LIN {X 0,Y 208.668,Z 381.617,A -85,B 0,C 180,E1 -22016.518,E2 -22016.518} C_VEL
LIN {X 0,Y 207.654,Z 387.475,A -85,B 0,C 180,E1 -22016.591,E2 -22016.591} C_VEL
LIN {X 0,Y 204.493,Z 399.145,A -85,B 0,C 180,E1 -22016.563,E2 -22016.563} C_VEL
LIN {X 0,Y 203.408,Z 405.081,A -85,B 0,C 180,E1 -22016.629,E2 -22016.629} C_VEL
LIN {X 0,Y 203.257,Z 407.077,A -85,B 0,C 180,E1 -22016.685,E2 -22016.685} C_VEL
LIN {X 0,Y 201.605,Z 442.654,A -85,B 0,C 180,E1 -22017.92,E2 -22017.92} C_VEL
LIN {X 0,Y 200.293,Z 456.074,A -85,B 0,C 180,E1 -22018.76,E2 -22018.76} C_VEL
LIN {X 0,Y 198.653,Z 468.006,A -85,B 0,C 180,E1 -22019.874,E2 -22019.874} C_VEL
LIN {X 0,Y 196.505,Z 480.066,A -85,B 0,C 180,E1 -22021.424,E2 -22021.424} C_VEL
LIN {X 0,Y 193.917,Z 491.578,A -85,B 0,C 180,E1 -22023.354,E2 -22023.354} C_VEL
LIN {X 0,Y 191.601,Z 501.991,A -85,B 0,C 180,E1 -22025.63,E2 -22025.63} C_VEL
LIN {X 0,Y 189.316,Z 511.311,A -85,B 0,C 180,E1 -22028.21,E2 -22028.21} C_VEL
LIN {X 0,Y 187.461,Z 518.995,A -85,B 0,C 180,E1 -22030.852,E2 -22030.852} C_VEL
LIN {X 0,Y 185.631,Z 526.51,A -85,B 0,C 180,E1 -22034.07,E2 -22034.07} C_VEL
LIN {X 0,Y 184.166,Z 533.424,A -85,B 0,C 180,E1 -22037.886,E2 -22037.886} C_VEL
LIN {X 0,Y 183.486,Z 537.971,A -85,B 0,C 180,E1 -22041.188,E2 -22041.188} C_VEL
LIN {X 0,Y 183.285,Z 540.362,A -85,B 0,C 180,E1 -22043.396,E2 -22043.396} C_VEL
LIN {X 0,Y 183.153,Z 542.708,A -85,B 0,C 180,E1 -22046.1,E2 -22046.1} C_VEL
LIN {X 0,Y 183.324,Z 544.894,A -85,B 0,C 180,E1 -22050.001,E2 -22050.001} C_VEL
LIN {X 0,Y 183.072,Z 545.742,A -85,B 0,C 180,E1 -22053.507,E2 -22053.507} C_VEL
LIN {X 0,Y 183.214,Z 545.668,A -85,B 0,C 180,E1 -22056.609,E2 -22056.609} C_VEL
LIN {X 0,Y 184.032,Z 544.175,A -85,B 0,C 180,E1 -22061.009,E2 -22061.009} C_VEL
LIN {X 0,Y 185.663,Z 541.115,A -85,B 0,C 180,E1 -22065.366,E2 -22065.366} C_VEL
LIN {X 0,Y 187.738,Z 537.669,A -85,B 0,C 180,E1 -22068.555,E2 -22068.555} C_VEL
LIN {X 0,Y 190.309,Z 533.167,A -85,B 0,C 180,E1 -22071.673,E2 -22071.673} C_VEL
LIN {X 0,Y 193.539,Z 527.136,A -85,B 0,C 180,E1 -22074.873,E2 -22074.873} C_VEL
LIN {X 0,Y 196.958,Z 520.396,A -85,B 0,C 180,E1 -22077.638,E2 -22077.638} C_VEL
LIN {X 0,Y 201.249,Z 511.587,A -85,B 0,C 180,E1 -22080.423,E2 -22080.423} C_VEL
LIN {X 0,Y 205.142,Z 502.581,A -85,B 0,C 180,E1 -22082.656,E2 -22082.656} C_VEL
LIN {X 0,Y 208.987,Z 492.681,A -85,B 0,C 180,E1 -22084.576,E2 -22084.576} C_VEL
LIN {X 0,Y 212.638,Z 481.706,A -85,B 0,C 180,E1 -22086.214,E2 -22086.214} C_VEL
LIN {X 0,Y 215.466,Z 471.415,A -85,B 0,C 180,E1 -22087.41,E2 -22087.41} C_VEL
LIN {X 0,Y 218.344,Z 458.36,A -85,B 0,C 180,E1 -22088.522,E2 -22088.522} C_VEL
LIN {X 0,Y 220.277,Z 445.531,A -85,B 0,C 180,E1 -22089.282,E2 -22089.282} C_VEL
LIN {X 0,Y 221.553,Z 429.787,A -85,B 0,C 180,E1 -22089.834,E2 -22089.834} C_VEL
LIN {X 0,Y 223.363,Z 398.956,A -85,B 0,C 180,E1 -22090.749,E2 -22090.749} C_VEL
LIN {X 0,Y 222.537,Z 393.348,A -85,B 0,C 180,E1 -22091.214,E2 -22091.214} C_VEL
LIN {X 0,Y 216.187,Z 378.63,A -85,B 0,C 180,E1 -22093.651,E2 -22093.651} C_VEL
LIN {X 0,Y 210.751,Z 367.719,A -85,B 0,C 180,E1 -22095.876,E2 -22095.876} C_VEL
LIN {X 0,Y 204.884,Z 357.45,A -85,B 0,C 180,E1 -22098.458,E2 -22098.458} C_VEL
LIN {X 0,Y 201.95,Z 352.743,A -85,B 0,C 180,E1 -22099.843,E2 -22099.843} C_VEL
LIN {X 0,Y 198.712,Z 347.595,A -85,B 0,C 180,E1 -22101.478,E2 -22101.478} C_VEL
LIN {X 0,Y 195.305,Z 342.411,A -85,B 0,C 180,E1 -22103.324,E2 -22103.324} C_VEL
LIN {X 0,Y 191.41,Z 336.757,A -85,B 0,C 180,E1 -22105.63,E2 -22105.63} C_VEL
LIN {X 0,Y 187.73,Z 332.249,A -85,B 0,C 180,E1 -22108,E2 -22108} C_VEL
LIN {X 0,Y 186.391,Z 329.867,A -85,B 0,C 180,E1 -22109.087,E2 -22109.087} C_VEL
LIN {X 0,Y 185.613,Z 327.361,A -85,B 0,C 180,E1 -22111.905,E2 -22111.905} C_VEL
LIN {X 0,Y 185.59,Z 327.368,A -85,B 0,C 180,E1 -22115.383,E2 -22115.383} C_VEL
LIN {X 0,Y 185.677,Z 327.344,A -85,B 0,C 180,E1 -22121.133,E2 -22121.133} C_VEL
LIN {X 0,Y 185.697,Z 327.342,A -85,B 0,C 180,E1 -22124.637,E2 -22124.637} C_VEL
LIN {X 0,Y 185.891,Z 327.313,A -85,B 0,C 180,E1 -22129.417,E2 -22129.417} C_VEL
LIN {X 0,Y 185.953,Z 327.306,A -85,B 0,C 180,E1 -22133.489,E2 -22133.489} C_VEL
LIN {X 0,Y 186.208,Z 327.274,A -85,B 0,C 180,E1 -22137.837,E2 -22137.837} C_VEL
LIN {X 0,Y 186.406,Z 327.249,A -85,B 0,C 180,E1 -22140,E2 -22140} C_VEL
LIN {X 0,Y 185.924,Z 327.309,A -85,B 0,C 180,E1 -22144.335,E2 -22144.335} C_VEL
LIN {X 0,Y 186.011,Z 327.3,A -85,B 0,C 180,E1 -22148.692,E2 -22148.692} C_VEL
LIN {X 0,Y 185.736,Z 327.337,A -85,B 0,C 180,E1 -22153.122,E2 -22153.122} C_VEL
LIN {X 0,Y 185.691,Z 327.346,A -85,B 0,C 180,E1 -22157.625,E2 -22157.625} C_VEL
LIN {X 0,Y 185.604,Z 327.548,A -85,B 0,C 180,E1 -22160.865,E2 -22160.865} C_VEL
LIN {X 0,Y 186.322,Z 329.769,A -85,B 0,C 180,E1 -22161.505,E2 -22161.505} C_VEL
LIN {X 0,Y 188.182,Z 332.015,A -85,B 0,C 180,E1 -22162.797,E2 -22162.797} C_VEL
LIN {X 0,Y 190.075,Z 333.259,A -85,B 0,C 180,E1 -22163.952,E2 -22163.952} C_VEL
LIN {X 0,Y 191.863,Z 336.387,A -85,B 0,C 180,E1 -22165.13,E2 -22165.13} C_VEL
LIN {X 0,Y 194.423,Z 338.858,A -85,B 0,C 180,E1 -22166.572,E2 -22166.572} C_VEL
LIN {X 0,Y 196.875,Z 342.368,A -85,B 0,C 180,E1 -22167.939,E2 -22167.939} C_VEL
LIN {X 0,Y 198.391,Z 344.088,A -85,B 0,C 180,E1 -22168.715,E2 -22168.715} C_VEL
LIN {X 0,Y 202.124,Z 349.183,A -85,B 0,C 180,E1 -22170.565,E2 -22170.565} C_VEL
LIN {X 0,Y 207.219,Z 356.189,A -85,B 0,C 180,E1 -22172.864,E2 -22172.864} C_VEL
LIN {X 0,Y 214.375,Z 367.343,A -85,B 0,C 180,E1 -22175.802,E2 -22175.802} C_VEL
LIN {X 0,Y 218.893,Z 375.323,A -85,B 0,C 180,E1 -22177.519,E2 -22177.519} C_VEL
LIN {X 0,Y 223.957,Z 386.107,A -85,B 0,C 180,E1 -22179.382,E2 -22179.382} C_VEL
LIN {X 0,Y 221.263,Z 429.958,A -85,B 0,C 180,E1 -22180.737,E2 -22180.737} C_VEL
LIN {X 0,Y 219.571,Z 443.344,A -85,B 0,C 180,E1 -22181.471,E2 -22181.471} C_VEL
LIN {X 0,Y 217.663,Z 453.695,A -85,B 0,C 180,E1 -22182.29,E2 -22182.29} C_VEL
LIN {X 0,Y 215.148,Z 465.009,A -85,B 0,C 180,E1 -22183.519,E2 -22183.519} C_VEL
LIN {X 0,Y 212.177,Z 475.253,A -85,B 0,C 180,E1 -22184.926,E2 -22184.926} C_VEL
LIN {X 0,Y 208.834,Z 485.292,A -85,B 0,C 180,E1 -22186.709,E2 -22186.709} C_VEL
LIN {X 0,Y 205.109,Z 494.662,A -85,B 0,C 180,E1 -22188.796,E2 -22188.796} C_VEL
LIN {X 0,Y 200.69,Z 504.369,A -85,B 0,C 180,E1 -22191.567,E2 -22191.567} C_VEL
LIN {X 0,Y 196.696,Z 512.209,A -85,B 0,C 180,E1 -22194.505,E2 -22194.505} C_VEL
LIN {X 0,Y 193.786,Z 517.529,A -85,B 0,C 180,E1 -22197.043,E2 -22197.043} C_VEL
LIN {X 0,Y 190.747,Z 522.64,A -85,B 0,C 180,E1 -22200.171,E2 -22200.171} C_VEL
LIN {X 0,Y 187.947,Z 527.003,A -85,B 0,C 180,E1 -22203.824,E2 -22203.824} C_VEL
LIN {X 0,Y 185.701,Z 530.147,A -85,B 0,C 180,E1 -22207.761,E2 -22207.761} C_VEL
LIN {X 0,Y 184.78,Z 531.287,A -85,B 0,C 180,E1 -22209.981,E2 -22209.981} C_VEL
LIN {X 0,Y 183.972,Z 532.088,A -85,B 0,C 180,E1 -22212.752,E2 -22212.752} C_VEL
LIN {X 0,Y 183.211,Z 532.19,A -85,B 0,C 180,E1 -22216.692,E2 -22216.692} C_VEL
LIN {X 0,Y 183.023,Z 531.678,A -85,B 0,C 180,E1 -22218.93,E2 -22218.93} C_VEL
LIN {X 0,Y 183,Z 530.746,A -85,B 0,C 180,E1 -22221.162,E2 -22221.162} C_VEL
LIN {X 0,Y 183.409,Z 528.14,A -85,B 0,C 180,E1 -22225.057,E2 -22225.057} C_VEL
LIN {X 0,Y 183.952,Z 524.248,A -85,B 0,C 180,E1 -22228.904,E2 -22228.904} C_VEL
LIN {X 0,Y 184.943,Z 519.717,A -85,B 0,C 180,E1 -22232.177,E2 -22232.177} C_VEL
LIN {X 0,Y 186.489,Z 512.867,A -85,B 0,C 180,E1 -22235.947,E2 -22235.947} C_VEL
LIN {X 0,Y 188.412,Z 505.439,A -85,B 0,C 180,E1 -22239.12,E2 -22239.12} C_VEL
LIN {X 0,Y 190.372,Z 497.865,A -85,B 0,C 180,E1 -22241.714,E2 -22241.714} C_VEL
LIN {X 0,Y 192.63,Z 488.695,A -85,B 0,C 180,E1 -22244.256,E2 -22244.256} C_VEL
LIN {X 0,Y 194.994,Z 478.471,A -85,B 0,C 180,E1 -22246.488,E2 -22246.488} C_VEL
LIN {X 0,Y 197.452,Z 467.103,A -85,B 0,C 180,E1 -22248.413,E2 -22248.413} C_VEL
LIN {X 0,Y 199.305,Z 455.369,A -85,B 0,C 180,E1 -22249.973,E2 -22249.973} C_VEL
LIN {X 0,Y 200.678,Z 442.511,A -85,B 0,C 180,E1 -22251.237,E2 -22251.237} C_VEL
LIN {X 0,Y 201.914,Z 429.718,A -85,B 0,C 180,E1 -22252.039,E2 -22252.039} C_VEL
LIN {X 0,Y 203.605,Z 395.641,A -85,B 0,C 180,E1 -22253.214,E2 -22253.214} C_VEL
LIN {X 0,Y 204.769,Z 366.988,A -85,B 0,C 180,E1 -22254.17,E2 -22254.17} C_VEL
LIN {X 0,Y 200.862,Z 356.621,A -85,B 0,C 180,E1 -22255.245,E2 -22255.245} C_VEL
LIN {X 0,Y 193.205,Z 341.376,A -85,B 0,C 180,E1 -22257.295,E2 -22257.295} C_VEL
LIN {X 0,Y 187.089,Z 330.978,A -85,B 0,C 180,E1 -22259.007,E2 -22259.007} C_VEL
LIN {X 0,Y 185.79,Z 328.546,A -85,B 0,C 180,E1 -22259.4,E2 -22259.4} C_VEL
LIN {X 0,Y 185.544,Z 327.369,A -85,B 0,C 180,E1 -22259.575,E2 -22259.575} C_VEL
LIN {X 0,Y 185.494,Z 327.378,A -85,B 0,C 180,E1 -22264.631,E2 -22264.631} C_VEL
LIN {X 0,Y 185.497,Z 327.373,A -85,B 0,C 180,E1 -22267.313,E2 -22267.313} C_VEL
LIN {X 0,Y 185.458,Z 327.383,A -85,B 0,C 180,E1 -22270.72,E2 -22270.72} C_VEL
LIN {X 0,Y 185.454,Z 327.379,A -85,B 0,C 180,E1 -22276.054,E2 -22276.054} C_VEL
LIN {X 0,Y 185.462,Z 327.371,A -85,B 0,C 180,E1 -22279.894,E2 -22279.894} C_VEL
LIN {X 0,Y 185.501,Z 327.364,A -85,B 0,C 180,E1 -22282.711,E2 -22282.711} C_VEL
LIN {X 0,Y 185.537,Z 327.362,A -85,B 0,C 180,E1 -22287.974,E2 -22287.974} C_VEL
LIN {X 0,Y 185.575,Z 327.347,A -85,B 0,C 180,E1 -22290.576,E2 -22290.576} C_VEL
LIN {X 0,Y 185.575,Z 327.37,A -85,B 0,C 180,E1 -22295.381,E2 -22295.381} C_VEL
LIN {X 0,Y 185.668,Z 327.34,A -85,B 0,C 180,E1 -22301.134,E2 -22301.134} C_VEL
LIN {X 0,Y 185.689,Z 327.354,A -85,B 0,C 180,E1 -22304.637,E2 -22304.637} C_VEL
LIN {X 0,Y 185.883,Z 327.307,A -85,B 0,C 180,E1 -22309.419,E2 -22309.419} C_VEL
LIN {X 0,Y 185.934,Z 327.319,A -85,B 0,C 180,E1 -22313.489,E2 -22313.489} C_VEL
LIN {X 0,Y 186.198,Z 327.283,A -85,B 0,C 180,E1 -22317.837,E2 -22317.837} C_VEL
LIN {X 0,Y 186.398,Z 327.242,A -85,B 0,C 180,E1 -22320,E2 -22320} C_VEL
LIN {X 0,Y 185.917,Z 327.323,A -85,B 0,C 180,E1 -22324.336,E2 -22324.336} C_VEL
LIN {X 0,Y 186.003,Z 327.303,A -85,B 0,C 180,E1 -22328.693,E2 -22328.693} C_VEL
LIN {X 0,Y 185.729,Z 327.338,A -85,B 0,C 180,E1 -22333.123,E2 -22333.123} C_VEL
LIN {X 0,Y 185.685,Z 327.35,A -85,B 0,C 180,E1 -22337.626,E2 -22337.626} C_VEL
LIN {X 0,Y 185.592,Z 327.363,A -85,B 0,C 180,E1 -22342.252,E2 -22342.252} C_VEL
LIN {X 0,Y 185.558,Z 327.37,A -85,B 0,C 180,E1 -22347.033,E2 -22347.033} C_VEL
LIN {X 0,Y 185.575,Z 327.368,A -85,B 0,C 180,E1 -22349.494,E2 -22349.494} C_VEL
LIN {X 0,Y 185.507,Z 327.38,A -85,B 0,C 180,E1 -22354.631,E2 -22354.631} C_VEL
LIN {X 0,Y 185.541,Z 327.375,A -85,B 0,C 180,E1 -22357.305,E2 -22357.305} C_VEL
LIN {X 0,Y 185.481,Z 327.384,A -85,B 0,C 180,E1 -22360.731,E2 -22360.731} C_VEL
LIN {X 0,Y 185.456,Z 327.387,A -85,B 0,C 180,E1 -22366.057,E2 -22366.057} C_VEL
LIN {X 0,Y 185.503,Z 327.579,A -85,B 0,C 180,E1 -22367.706,E2 -22367.706} C_VEL
LIN {X 0,Y 186.847,Z 332.585,A -85,B 0,C 180,E1 -22370.517,E2 -22370.517} C_VEL
LIN {X 0,Y 193.158,Z 346.017,A -85,B 0,C 180,E1 -22372.399,E2 -22372.399} C_VEL
LIN {X 0,Y 200.302,Z 363.714,A -85,B 0,C 180,E1 -22374.448,E2 -22374.448} C_VEL
LIN {X 0,Y 201.381,Z 367.117,A -85,B 0,C 180,E1 -22374.772,E2 -22374.772} C_VEL
LIN {X 0,Y 203.856,Z 392.612,A -85,B 0,C 180,E1 -22376.204,E2 -22376.204} C_VEL
LIN {X 0,Y 203.257,Z 407.077,A -85,B 0,C 180,E1 -22376.685,E2 -22376.685} C_VEL
LIN {X 0,Y 202.421,Z 412.922,A -85,B 0,C 180,E1 -22376.783,E2 -22376.783} C_VEL
LIN {X 0,Y 196.521,Z 431.869,A -85,B 0,C 180,E1 -22376.609,E2 -22376.609} C_VEL
LIN {X 0,Y 195.694,Z 437.696,A -85,B 0,C 180,E1 -22376.747,E2 -22376.747} C_VEL
LIN {X 0,Y 194.622,Z 450.72,A -85,B 0,C 180,E1 -22377.435,E2 -22377.435} C_VEL
LIN {X 0,Y 192.985,Z 462.95,A -85,B 0,C 180,E1 -22378.435,E2 -22378.435} C_VEL
LIN {X 0,Y 191.223,Z 473.552,A -85,B 0,C 180,E1 -22379.647,E2 -22379.647} C_VEL
LIN {X 0,Y 188.881,Z 485.038,A -85,B 0,C 180,E1 -22381.378,E2 -22381.378} C_VEL
LIN {X 0,Y 186.426,Z 495.503,A -85,B 0,C 180,E1 -22383.407,E2 -22383.407} C_VEL
LIN {X 0,Y 184.119,Z 505.106,A -85,B 0,C 180,E1 -22385.776,E2 -22385.776} C_VEL
LIN {X 0,Y 181.706,Z 514.437,A -85,B 0,C 180,E1 -22388.669,E2 -22388.669} C_VEL
LIN {X 0,Y 179.712,Z 522.324,A -85,B 0,C 180,E1 -22391.77,E2 -22391.77} C_VEL
LIN {X 0,Y 177.949,Z 529.121,A -85,B 0,C 180,E1 -22395.126,E2 -22395.126} C_VEL
LIN {X 0,Y 176.885,Z 534.552,A -85,B 0,C 180,E1 -22398.543,E2 -22398.543} C_VEL
LIN {X 0,Y 176.309,Z 538.777,A -85,B 0,C 180,E1 -22401.981,E2 -22401.981} C_VEL
LIN {X 0,Y 176.067,Z 542.57,A -85,B 0,C 180,E1 -22406.305,E2 -22406.305} C_VEL
LIN {X 0,Y 176.224,Z 544.569,A -85,B 0,C 180,E1 -22410.001,E2 -22410.001} C_VEL
LIN {X 0,Y 175.992,Z 545.429,A -85,B 0,C 180,E1 -22413.293,E2 -22413.293} C_VEL
LIN {X 0,Y 176.141,Z 545.416,A -85,B 0,C 180,E1 -22416.876,E2 -22416.876} C_VEL
LIN {X 0,Y 176.473,Z 544.913,A -85,B 0,C 180,E1 -22419.167,E2 -22419.167} C_VEL
LIN {X 0,Y 177.798,Z 542.685,A -85,B 0,C 180,E1 -22423.721,E2 -22423.721} C_VEL
LIN {X 0,Y 179.472,Z 539.95,A -85,B 0,C 180,E1 -22427.08,E2 -22427.08} C_VEL
LIN {X 0,Y 181.836,Z 536.221,A -85,B 0,C 180,E1 -22430.357,E2 -22430.357} C_VEL
LIN {X 0,Y 184.785,Z 531.399,A -85,B 0,C 180,E1 -22433.538,E2 -22433.538} C_VEL
LIN {X 0,Y 188.699,Z 524.227,A -85,B 0,C 180,E1 -22437.146,E2 -22437.146} C_VEL
LIN {X 0,Y 192.861,Z 516.414,A -85,B 0,C 180,E1 -22440.071,E2 -22440.071} C_VEL
LIN {X 0,Y 197.537,Z 506.693,A -85,B 0,C 180,E1 -22442.859,E2 -22442.859} C_VEL
LIN {X 0,Y 201.873,Z 496.64,A -85,B 0,C 180,E1 -22445.061,E2 -22445.061} C_VEL
LIN {X 0,Y 205.535,Z 486.698,A -85,B 0,C 180,E1 -22446.755,E2 -22446.755} C_VEL
LIN {X 0,Y 208.901,Z 475.911,A -85,B 0,C 180,E1 -22448.184,E2 -22448.184} C_VEL
LIN {X 0,Y 212.165,Z 463.039,A -85,B 0,C 180,E1 -22449.446,E2 -22449.446} C_VEL
LIN {X 0,Y 214.523,Z 450.272,A -85,B 0,C 180,E1 -22450.321,E2 -22450.321} C_VEL
LIN {X 0,Y 215.99,Z 437.281,A -85,B 0,C 180,E1 -22450.902,E2 -22450.902} C_VEL
LIN {X 0,Y 218.297,Z 399.597,A -85,B 0,C 180,E1 -22452.056,E2 -22452.056} C_VEL
LIN {X 0,Y 217.661,Z 396.23,A -85,B 0,C 180,E1 -22452.389,E2 -22452.389} C_VEL
LIN {X 0,Y 212.018,Z 382.834,A -85,B 0,C 180,E1 -22454.696,E2 -22454.696} C_VEL
LIN {X 0,Y 206.837,Z 372.266,A -85,B 0,C 180,E1 -22456.94,E2 -22456.94} C_VEL
LIN {X 0,Y 201.153,Z 362.114,A -85,B 0,C 180,E1 -22459.595,E2 -22459.595} C_VEL
LIN {X 0,Y 195.872,Z 353.361,A -85,B 0,C 180,E1 -22462.339,E2 -22462.339} C_VEL
LIN {X 0,Y 192.294,Z 347.95,A -85,B 0,C 180,E1 -22464.374,E2 -22464.374} C_VEL
LIN {X 0,Y 188.323,Z 342.052,A -85,B 0,C 180,E1 -22466.882,E2 -22466.882} C_VEL
LIN {X 0,Y 185.387,Z 338.281,A -85,B 0,C 180,E1 -22468.9,E2 -22468.9} C_VEL
LIN {X 0,Y 184.061,Z 336.139,A -85,B 0,C 180,E1 -22469.923,E2 -22469.923} C_VEL
LIN {X 0,Y 180.807,Z 332.628,A -85,B 0,C 180,E1 -22472.51,E2 -22472.51} C_VEL
LIN {X 0,Y 179.066,Z 330.245,A -85,B 0,C 180,E1 -22474.11,E2 -22474.11} C_VEL
LIN {X 0,Y 178.701,Z 329.199,A -85,B 0,C 180,E1 -22474.58,E2 -22474.58} C_VEL
LIN {X 0,Y 178.551,Z 328.24,A -85,B 0,C 180,E1 -22475.8,E2 -22475.8} C_VEL
LIN {X 0,Y 178.652,Z 328.218,A -85,B 0,C 180,E1 -22481.656,E2 -22481.656} C_VEL
LIN {X 0,Y 178.66,Z 328.216,A -85,B 0,C 180,E1 -22486.348,E2 -22486.348} C_VEL
LIN {X 0,Y 178.916,Z 328.183,A -85,B 0,C 180,E1 -22490.96,E2 -22490.96} C_VEL
LIN {X 0,Y 178.869,Z 328.188,A -85,B 0,C 180,E1 -22495.493,E2 -22495.493} C_VEL
LIN {X 0,Y 179.369,Z 328.125,A -85,B 0,C 180,E1 -22500,E2 -22500} C_VEL
LIN {X 0,Y 178.873,Z 328.188,A -85,B 0,C 180,E1 -22504.507,E2 -22504.507} C_VEL
LIN {X 0,Y 178.961,Z 328.18,A -85,B 0,C 180,E1 -22509.037,E2 -22509.037} C_VEL
LIN {X 0,Y 178.643,Z 328.231,A -85,B 0,C 180,E1 -22514.816,E2 -22514.816} C_VEL
LIN {X 0,Y 178.65,Z 328.221,A -85,B 0,C 180,E1 -22515.838,E2 -22515.838} C_VEL
LIN {X 0,Y 179.298,Z 330.501,A -85,B 0,C 180,E1 -22516.656,E2 -22516.656} C_VEL
LIN {X 0,Y 181.357,Z 332.992,A -85,B 0,C 180,E1 -22518.482,E2 -22518.482} C_VEL
LIN {X 0,Y 183.341,Z 334.22,A -85,B 0,C 180,E1 -22519.981,E2 -22519.981} C_VEL
LIN {X 0,Y 184.972,Z 337.251,A -85,B 0,C 180,E1 -22521.304,E2 -22521.304} C_VEL
LIN {X 0,Y 187.798,Z 339.829,A -85,B 0,C 180,E1 -22523.201,E2 -22523.201} C_VEL
LIN {X 0,Y 189.939,Z 343.067,A -85,B 0,C 180,E1 -22524.625,E2 -22524.625} C_VEL
LIN {X 0,Y 191.9,Z 345.056,A -85,B 0,C 180,E1 -22525.779,E2 -22525.779} C_VEL
LIN {X 0,Y 194.511,Z 348.679,A -85,B 0,C 180,E1 -22527.285,E2 -22527.285} C_VEL
LIN {X 0,Y 196.108,Z 350.769,A -85,B 0,C 180,E1 -22528.149,E2 -22528.149} C_VEL
LIN {X 0,Y 199.235,Z 355.011,A -85,B 0,C 180,E1 -22529.757,E2 -22529.757} C_VEL
LIN {X 0,Y 204.041,Z 361.893,A -85,B 0,C 180,E1 -22532.04,E2 -22532.04} C_VEL
LIN {X 0,Y 210.975,Z 372.89,A -85,B 0,C 180,E1 -22535.019,E2 -22535.019} C_VEL
LIN {X 0,Y 215.078,Z 380.406,A -85,B 0,C 180,E1 -22536.663,E2 -22536.663} C_VEL
LIN {X 0,Y 218.932,Z 388.801,A -85,B 0,C 180,E1 -22538.166,E2 -22538.166} C_VEL
LIN {X 0,Y 216.251,Z 429.585,A -85,B 0,C 180,E1 -22539.412,E2 -22539.412} C_VEL
LIN {X 0,Y 214.496,Z 443.281,A -85,B 0,C 180,E1 -22540.163,E2 -22540.163} C_VEL
LIN {X 0,Y 212.721,Z 452.374,A -85,B 0,C 180,E1 -22540.848,E2 -22540.848} C_VEL
LIN {X 0,Y 210.09,Z 464.281,A -85,B 0,C 180,E1 -22542.134,E2 -22542.134} C_VEL
LIN {X 0,Y 206.641,Z 475.81,A -85,B 0,C 180,E1 -22543.719,E2 -22543.719} C_VEL
LIN {X 0,Y 202.748,Z 486.875,A -85,B 0,C 180,E1 -22545.764,E2 -22545.764} C_VEL
LIN {X 0,Y 198.177,Z 497.542,A -85,B 0,C 180,E1 -22548.283,E2 -22548.283} C_VEL
LIN {X 0,Y 194.287,Z 505.511,A -85,B 0,C 180,E1 -22550.725,E2 -22550.725} C_VEL
LIN {X 0,Y 190.137,Z 513.157,A -85,B 0,C 180,E1 -22553.742,E2 -22553.742} C_VEL
LIN {X 0,Y 186.554,Z 519.263,A -85,B 0,C 180,E1 -22556.889,E2 -22556.889} C_VEL
LIN {X 0,Y 183.474,Z 524.057,A -85,B 0,C 180,E1 -22560.133,E2 -22560.133} C_VEL
LIN {X 0,Y 181.198,Z 527.369,A -85,B 0,C 180,E1 -22563.136,E2 -22563.136} C_VEL
LIN {X 0,Y 178.969,Z 530.268,A -85,B 0,C 180,E1 -22566.877,E2 -22566.877} C_VEL
LIN {X 0,Y 177.946,Z 531.462,A -85,B 0,C 180,E1 -22569.178,E2 -22569.178} C_VEL
LIN {X 0,Y 176.937,Z 532.38,A -85,B 0,C 180,E1 -22572.418,E2 -22572.418} C_VEL
LIN {X 0,Y 176.18,Z 532.475,A -85,B 0,C 180,E1 -22576.151,E2 -22576.151} C_VEL
LIN {X 0,Y 175.943,Z 532.023,A -85,B 0,C 180,E1 -22578.478,E2 -22578.478} C_VEL
LIN {X 0,Y 175.907,Z 531.128,A -85,B 0,C 180,E1 -22580.803,E2 -22580.803} C_VEL
LIN {X 0,Y 176.322,Z 528.33,A -85,B 0,C 180,E1 -22585.185,E2 -22585.185} C_VEL
LIN {X 0,Y 176.859,Z 524.762,A -85,B 0,C 180,E1 -22588.86,E2 -22588.86} C_VEL
LIN {X 0,Y 177.844,Z 520.309,A -85,B 0,C 180,E1 -22592.264,E2 -22592.264} C_VEL
LIN {X 0,Y 179.443,Z 513.58,A -85,B 0,C 180,E1 -22596.182,E2 -22596.182} C_VEL
LIN {X 0,Y 181.422,Z 506.248,A -85,B 0,C 180,E1 -22599.475,E2 -22599.475} C_VEL
LIN {X 0,Y 183.885,Z 497.15,A -85,B 0,C 180,E1 -22602.694,E2 -22602.694} C_VEL
LIN {X 0,Y 186.583,Z 486.625,A -85,B 0,C 180,E1 -22605.566,E2 -22605.566} C_VEL
LIN {X 0,Y 189.131,Z 475.903,A -85,B 0,C 180,E1 -22607.851,E2 -22607.851} C_VEL
LIN {X 0,Y 191.467,Z 465.446,A -85,B 0,C 180,E1 -22609.568,E2 -22609.568} C_VEL
LIN {X 0,Y 193.287,Z 453.009,A -85,B 0,C 180,E1 -22611.181,E2 -22611.181} C_VEL
LIN {X 0,Y 194.656,Z 439.934,A -85,B 0,C 180,E1 -22612.416,E2 -22612.416} C_VEL
LIN {X 0,Y 195.857,Z 427.878,A -85,B 0,C 180,E1 -22613.107,E2 -22613.107} C_VEL
LIN {X 0,Y 198.598,Z 368.674,A -85,B 0,C 180,E1 -22615.139,E2 -22615.139} C_VEL
LIN {X 0,Y 195.296,Z 359.966,A -85,B 0,C 180,E1 -22616.096,E2 -22616.096} C_VEL
LIN {X 0,Y 188.027,Z 345.386,A -85,B 0,C 180,E1 -22618.151,E2 -22618.151} C_VEL
LIN {X 0,Y 180.377,Z 332.254,A -85,B 0,C 180,E1 -22620.442,E2 -22620.442} C_VEL
LIN {X 0,Y 178.842,Z 329.74,A -85,B 0,C 180,E1 -22620.928,E2 -22620.928} C_VEL
LIN {X 0,Y 178.491,Z 328.248,A -85,B 0,C 180,E1 -22621.116,E2 -22621.116} C_VEL
LIN {X 0,Y 178.48,Z 328.252,A -85,B 0,C 180,E1 -22624.217,E2 -22624.217} C_VEL
LIN {X 0,Y 178.384,Z 328.255,A -85,B 0,C 180,E1 -22629.075,E2 -22629.075} C_VEL
LIN {X 0,Y 178.389,Z 328.262,A -85,B 0,C 180,E1 -22632.045,E2 -22632.045} C_VEL
LIN {X 0,Y 178.388,Z 328.25,A -85,B 0,C 180,E1 -22635.163,E2 -22635.163} C_VEL
LIN {X 0,Y 178.398,Z 328.26,A -85,B 0,C 180,E1 -22638.458,E2 -22638.458} C_VEL
LIN {X 0,Y 178.417,Z 328.253,A -85,B 0,C 180,E1 -22643.782,E2 -22643.782} C_VEL
LIN {X 0,Y 178.481,Z 328.249,A -85,B 0,C 180,E1 -22646.546,E2 -22646.546} C_VEL
LIN {X 0,Y 178.517,Z 328.224,A -85,B 0,C 180,E1 -22650.007,E2 -22650.007} C_VEL
LIN {X 0,Y 178.515,Z 328.248,A -85,B 0,C 180,E1 -22654.885,E2 -22654.885} C_VEL
LIN {X 0,Y 178.616,Z 328.214,A -85,B 0,C 180,E1 -22660.786,E2 -22660.786} C_VEL
LIN {X 0,Y 178.652,Z 328.227,A -85,B 0,C 180,E1 -22666.348,E2 -22666.348} C_VEL
LIN {X 0,Y 178.901,Z 328.176,A -85,B 0,C 180,E1 -22670.96,E2 -22670.96} C_VEL
LIN {X 0,Y 179.144,Z 328.161,A -85,B 0,C 180,E1 -22677.752,E2 -22677.752} C_VEL
LIN {X 0,Y 179.362,Z 328.117,A -85,B 0,C 180,E1 -22680,E2 -22680} C_VEL
LIN {X 0,Y 178.866,Z 328.202,A -85,B 0,C 180,E1 -22684.507,E2 -22684.507} C_VEL
LIN {X 0,Y 178.954,Z 328.179,A -85,B 0,C 180,E1 -22689.038,E2 -22689.038} C_VEL
LIN {X 0,Y 178.655,Z 328.224,A -85,B 0,C 180,E1 -22693.653,E2 -22693.653} C_VEL
LIN {X 0,Y 178.619,Z 328.235,A -85,B 0,C 180,E1 -22699.217,E2 -22699.217} C_VEL
LIN {X 0,Y 178.53,Z 328.246,A -85,B 0,C 180,E1 -22705.125,E2 -22705.125} C_VEL
LIN {X 0,Y 178.475,Z 328.253,A -85,B 0,C 180,E1 -22710.792,E2 -22710.792} C_VEL
LIN {X 0,Y 178.488,Z 328.254,A -85,B 0,C 180,E1 -22714.224,E2 -22714.224} C_VEL
LIN {X 0,Y 178.415,Z 328.264,A -85,B 0,C 180,E1 -22719.07,E2 -22719.07} C_VEL
LIN {X 0,Y 178.399,Z 328.267,A -85,B 0,C 180,E1 -22722.045,E2 -22722.045} C_VEL
LIN {X 0,Y 178.447,Z 328.398,A -85,B 0,C 180,E1 -22726.55,E2 -22726.55} C_VEL
LIN {X 0,Y 179.452,Z 332.198,A -85,B 0,C 180,E1 -22728.823,E2 -22728.823} C_VEL
LIN {X 0,Y 186.235,Z 346.009,A -85,B 0,C 180,E1 -22731.006,E2 -22731.006} C_VEL
LIN {X 0,Y 192.201,Z 360.384,A -85,B 0,C 180,E1 -22732.843,E2 -22732.843} C_VEL
LIN {X 0,Y 195.432,Z 369.201,A -85,B 0,C 180,E1 -22733.82,E2 -22733.82} C_VEL
LIN {X 0,Y 197.665,Z 392.61,A -85,B 0,C 180,E1 -22735.192,E2 -22735.192} C_VEL
LIN {X 0,Y 195.694,Z 437.696,A -85,B 0,C 180,E1 -22736.747,E2 -22736.747} C_VEL
LIN {X 0,Y 194.768,Z 443.493,A -85,B 0,C 180,E1 -22736.919,E2 -22736.919} C_VEL
LIN {X 0,Y 191.345,Z 452.775,A -85,B 0,C 180,E1 -22737.101,E2 -22737.101} C_VEL
LIN {X 0,Y 187.517,Z 461.874,A -85,B 0,C 180,E1 -22737.468,E2 -22737.468} C_VEL
LIN {X 0,Y 186.011,Z 467.368,A -85,B 0,C 180,E1 -22737.957,E2 -22737.957} C_VEL
LIN {X 0,Y 183.695,Z 479.212,A -85,B 0,C 180,E1 -22739.542,E2 -22739.542} C_VEL
LIN {X 0,Y 180.97,Z 490.796,A -85,B 0,C 180,E1 -22741.595,E2 -22741.595} C_VEL
LIN {X 0,Y 178.342,Z 501.248,A -85,B 0,C 180,E1 -22743.999,E2 -22743.999} C_VEL
LIN {X 0,Y 175.806,Z 510.875,A -85,B 0,C 180,E1 -22746.846,E2 -22746.846} C_VEL
LIN {X 0,Y 173.626,Z 519.02,A -85,B 0,C 180,E1 -22749.877,E2 -22749.877} C_VEL
LIN {X 0,Y 171.651,Z 526.44,A -85,B 0,C 180,E1 -22753.347,E2 -22753.347} C_VEL
LIN {X 0,Y 170.199,Z 532.376,A -85,B 0,C 180,E1 -22756.874,E2 -22756.874} C_VEL
LIN {X 0,Y 169.396,Z 537.048,A -85,B 0,C 180,E1 -22760.449,E2 -22760.449} C_VEL
LIN {X 0,Y 169.044,Z 540.587,A -85,B 0,C 180,E1 -22764.035,E2 -22764.035} C_VEL
LIN {X 0,Y 168.997,Z 543.093,A -85,B 0,C 180,E1 -22767.618,E2 -22767.618} C_VEL
LIN {X 0,Y 169.126,Z 544.244,A -85,B 0,C 180,E1 -22770.001,E2 -22770.001} C_VEL
LIN {X 0,Y 168.91,Z 545.056,A -85,B 0,C 180,E1 -22773.036,E2 -22773.036} C_VEL
LIN {X 0,Y 169.093,Z 545.163,A -85,B 0,C 180,E1 -22777.164,E2 -22777.164} C_VEL
LIN {X 0,Y 169.455,Z 544.701,A -85,B 0,C 180,E1 -22779.55,E2 -22779.55} C_VEL
LIN {X 0,Y 170.861,Z 542.529,A -85,B 0,C 180,E1 -22784.289,E2 -22784.289} C_VEL
LIN {X 0,Y 172.681,Z 539.846,A -85,B 0,C 180,E1 -22787.774,E2 -22787.774} C_VEL
LIN {X 0,Y 175.163,Z 536.172,A -85,B 0,C 180,E1 -22791.169,E2 -22791.169} C_VEL
LIN {X 0,Y 178.269,Z 531.41,A -85,B 0,C 180,E1 -22794.454,E2 -22794.454} C_VEL
LIN {X 0,Y 182.39,Z 524.302,A -85,B 0,C 180,E1 -22798.167,E2 -22798.167} C_VEL
LIN {X 0,Y 186.763,Z 516.601,A -85,B 0,C 180,E1 -22801.16,E2 -22801.16} C_VEL
LIN {X 0,Y 191.639,Z 506.97,A -85,B 0,C 180,E1 -22804.006,E2 -22804.006} C_VEL
LIN {X 0,Y 196.114,Z 497.051,A -85,B 0,C 180,E1 -22806.25,E2 -22806.25} C_VEL
LIN {X 0,Y 199.92,Z 487.29,A -85,B 0,C 180,E1 -22807.967,E2 -22807.967} C_VEL
LIN {X 0,Y 203.391,Z 476.72,A -85,B 0,C 180,E1 -22809.416,E2 -22809.416} C_VEL
LIN {X 0,Y 206.787,Z 464.046,A -85,B 0,C 180,E1 -22810.698,E2 -22810.698} C_VEL
LIN {X 0,Y 209.306,Z 451.47,A -85,B 0,C 180,E1 -22811.603,E2 -22811.603} C_VEL
LIN {X 0,Y 210.955,Z 438.305,A -85,B 0,C 180,E1 -22812.224,E2 -22812.224} C_VEL
LIN {X 0,Y 213.36,Z 400.947,A -85,B 0,C 180,E1 -22813.387,E2 -22813.387} C_VEL
LIN {X 0,Y 212.228,Z 397.427,A -85,B 0,C 180,E1 -22813.897,E2 -22813.897} C_VEL
LIN {X 0,Y 206.603,Z 384.131,A -85,B 0,C 180,E1 -22816.377,E2 -22816.377} C_VEL
LIN {X 0,Y 200.875,Z 372.749,A -85,B 0,C 180,E1 -22819.072,E2 -22819.072} C_VEL
LIN {X 0,Y 195.766,Z 363.764,A -85,B 0,C 180,E1 -22821.709,E2 -22821.709} C_VEL
LIN {X 0,Y 192.379,Z 358.177,A -85,B 0,C 180,E1 -22823.619,E2 -22823.619} C_VEL
LIN {X 0,Y 189.52,Z 353.627,A -85,B 0,C 180,E1 -22825.36,E2 -22825.36} C_VEL
LIN {X 0,Y 185.777,Z 347.996,A -85,B 0,C 180,E1 -22827.86,E2 -22827.86} C_VEL
LIN {X 0,Y 182.772,Z 343.723,A -85,B 0,C 180,E1 -22830.091,E2 -22830.091} C_VEL
LIN {X 0,Y 181.827,Z 342.306,A -85,B 0,C 180,E1 -22830.854,E2 -22830.854} C_VEL
LIN {X 0,Y 178.915,Z 339.044,A -85,B 0,C 180,E1 -22833.302,E2 -22833.302} C_VEL
LIN {X 0,Y 177.079,Z 336.345,A -85,B 0,C 180,E1 -22835.105,E2 -22835.105} C_VEL
LIN {X 0,Y 176.384,Z 335.102,A -85,B 0,C 180,E1 -22835.871,E2 -22835.871} C_VEL
LIN {X 0,Y 173.375,Z 333.129,A -85,B 0,C 180,E1 -22839.187,E2 -22839.187} C_VEL
LIN {X 0,Y 172.005,Z 330.762,A -85,B 0,C 180,E1 -22841.23,E2 -22841.23} C_VEL
LIN {X 0,Y 171.577,Z 329.101,A -85,B 0,C 180,E1 -22842.109,E2 -22842.109} C_VEL
LIN {X 0,Y 171.684,Z 329.092,A -85,B 0,C 180,E1 -22848.189,E2 -22848.189} C_VEL
LIN {X 0,Y 171.852,Z 329.061,A -85,B 0,C 180,E1 -22850.585,E2 -22850.585} C_VEL
LIN {X 0,Y 171.818,Z 329.065,A -85,B 0,C 180,E1 -22855.307,E2 -22855.307} C_VEL
LIN {X 0,Y 172.332,Z 329.001,A -85,B 0,C 180,E1 -22860,E2 -22860} C_VEL
LIN {X 0,Y 171.822,Z 329.067,A -85,B 0,C 180,E1 -22864.692,E2 -22864.692} C_VEL
LIN {X 0,Y 171.944,Z 329.12,A -85,B 0,C 180,E1 -22868.965,E2 -22868.965} C_VEL
LIN {X 0,Y 172.414,Z 331.1,A -85,B 0,C 180,E1 -22869.91,E2 -22869.91} C_VEL
LIN {X 0,Y 174.216,Z 333.714,A -85,B 0,C 180,E1 -22872.375,E2 -22872.375} C_VEL
LIN {X 0,Y 176.773,Z 335.233,A -85,B 0,C 180,E1 -22875.05,E2 -22875.05} C_VEL
LIN {X 0,Y 178.236,Z 338.115,A -85,B 0,C 180,E1 -22876.611,E2 -22876.611} C_VEL
LIN {X 0,Y 180.839,Z 340.462,A -85,B 0,C 180,E1 -22878.83,E2 -22878.83} C_VEL
LIN {X 0,Y 181.492,Z 341.215,A -85,B 0,C 180,E1 -22879.364,E2 -22879.364} C_VEL
LIN {X 0,Y 183.592,Z 344.388,A -85,B 0,C 180,E1 -22881.05,E2 -22881.05} C_VEL
LIN {X 0,Y 185.611,Z 346.276,A -85,B 0,C 180,E1 -22882.452,E2 -22882.452} C_VEL
LIN {X 0,Y 188.067,Z 349.743,A -85,B 0,C 180,E1 -22884.125,E2 -22884.125} C_VEL
LIN {X 0,Y 189.617,Z 351.552,A -85,B 0,C 180,E1 -22885.089,E2 -22885.089} C_VEL
LIN {X 0,Y 193.595,Z 356.997,A -85,B 0,C 180,E1 -22887.425,E2 -22887.425} C_VEL
LIN {X 0,Y 198.643,Z 364.059,A -85,B 0,C 180,E1 -22890.074,E2 -22890.074} C_VEL
LIN {X 0,Y 205.398,Z 374.695,A -85,B 0,C 180,E1 -22893.248,E2 -22893.248} C_VEL
LIN {X 0,Y 210.2,Z 383.175,A -85,B 0,C 180,E1 -22895.305,E2 -22895.305} C_VEL
LIN {X 0,Y 213.895,Z 391.197,A -85,B 0,C 180,E1 -22896.844,E2 -22896.844} C_VEL
LIN {X 0,Y 211.245,Z 430.465,A -85,B 0,C 180,E1 -22898.086,E2 -22898.086} C_VEL
LIN {X 0,Y 209.392,Z 444.021,A -85,B 0,C 180,E1 -22898.843,E2 -22898.843} C_VEL
LIN {X 0,Y 207.287,Z 454.406,A -85,B 0,C 180,E1 -22899.673,E2 -22899.673} C_VEL
LIN {X 0,Y 204.628,Z 465.542,A -85,B 0,C 180,E1 -22900.922,E2 -22900.922} C_VEL
LIN {X 0,Y 201.203,Z 476.359,A -85,B 0,C 180,E1 -22902.447,E2 -22902.447} C_VEL
LIN {X 0,Y 197.148,Z 487.365,A -85,B 0,C 180,E1 -22904.523,E2 -22904.523} C_VEL
LIN {X 0,Y 192.975,Z 496.738,A -85,B 0,C 180,E1 -22906.751,E2 -22906.751} C_VEL
LIN {X 0,Y 188.707,Z 505.21,A -85,B 0,C 180,E1 -22909.326,E2 -22909.326} C_VEL
LIN {X 0,Y 184.32,Z 512.974,A -85,B 0,C 180,E1 -22912.405,E2 -22912.405} C_VEL
LIN {X 0,Y 180.468,Z 519.166,A -85,B 0,C 180,E1 -22915.619,E2 -22915.619} C_VEL
LIN {X 0,Y 177.175,Z 524.037,A -85,B 0,C 180,E1 -22918.957,E2 -22918.957} C_VEL
LIN {X 0,Y 174.464,Z 527.745,A -85,B 0,C 180,E1 -22922.403,E2 -22922.403} C_VEL
LIN {X 0,Y 172.286,Z 530.391,A -85,B 0,C 180,E1 -22925.924,E2 -22925.924} C_VEL
LIN {X 0,Y 171.155,Z 531.621,A -85,B 0,C 180,E1 -22928.311,E2 -22928.311} C_VEL
LIN {X 0,Y 169.929,Z 532.669,A -85,B 0,C 180,E1 -22932.034,E2 -22932.034} C_VEL
LIN {X 0,Y 169.175,Z 532.76,A -85,B 0,C 180,E1 -22935.565,E2 -22935.565} C_VEL
LIN {X 0,Y 168.872,Z 532.348,A -85,B 0,C 180,E1 -22937.989,E2 -22937.989} C_VEL
LIN {X 0,Y 168.802,Z 531.509,A -85,B 0,C 180,E1 -22940.412,E2 -22940.412} C_VEL
LIN {X 0,Y 168.926,Z 530.247,A -85,B 0,C 180,E1 -22942.829,E2 -22942.829} C_VEL
LIN {X 0,Y 169.314,Z 527.97,A -85,B 0,C 180,E1 -22946.008,E2 -22946.008} C_VEL
LIN {X 0,Y 169.975,Z 523.944,A -85,B 0,C 180,E1 -22949.999,E2 -22949.999} C_VEL
LIN {X 0,Y 171.145,Z 519.179,A -85,B 0,C 180,E1 -22953.53,E2 -22953.53} C_VEL
LIN {X 0,Y 173.021,Z 512.058,A -85,B 0,C 180,E1 -22957.585,E2 -22957.585} C_VEL
LIN {X 0,Y 175.237,Z 504.284,A -85,B 0,C 180,E1 -22960.981,E2 -22960.981} C_VEL
LIN {X 0,Y 177.956,Z 494.571,A -85,B 0,C 180,E1 -22964.289,E2 -22964.289} C_VEL
LIN {X 0,Y 180.631,Z 484.5,A -85,B 0,C 180,E1 -22966.965,E2 -22966.965} C_VEL
LIN {X 0,Y 183.375,Z 473.076,A -85,B 0,C 180,E1 -22969.301,E2 -22969.301} C_VEL
LIN {X 0,Y 185.741,Z 461.851,A -85,B 0,C 180,E1 -22971.065,E2 -22971.065} C_VEL
LIN {X 0,Y 187.501,Z 449.331,A -85,B 0,C 180,E1 -22972.592,E2 -22972.592} C_VEL
LIN {X 0,Y 188.754,Z 437.732,A -85,B 0,C 180,E1 -22973.593,E2 -22973.593} C_VEL
LIN {X 0,Y 189.9,Z 424.557,A -85,B 0,C 180,E1 -22974.281,E2 -22974.281} C_VEL
LIN {X 0,Y 192.483,Z 370.279,A -85,B 0,C 180,E1 -22976.173,E2 -22976.173} C_VEL
LIN {X 0,Y 189.743,Z 363.228,A -85,B 0,C 180,E1 -22977.006,E2 -22977.006} C_VEL
LIN {X 0,Y 183.025,Z 349.577,A -85,B 0,C 180,E1 -22979.017,E2 -22979.017} C_VEL
LIN {X 0,Y 175.728,Z 336.947,A -85,B 0,C 180,E1 -22981.325,E2 -22981.325} C_VEL
LIN {X 0,Y 173.259,Z 333.051,A -85,B 0,C 180,E1 -22982.147,E2 -22982.147} C_VEL
LIN {X 0,Y 171.727,Z 330.466,A -85,B 0,C 180,E1 -22982.683,E2 -22982.683} C_VEL
LIN {X 0,Y 171.432,Z 329.128,A -85,B 0,C 180,E1 -22982.891,E2 -22982.891} C_VEL
LIN {X 0,Y 171.356,Z 329.13,A -85,B 0,C 180,E1 -22987.965,E2 -22987.965} C_VEL
LIN {X 0,Y 171.327,Z 329.137,A -85,B 0,C 180,E1 -22992.407,E2 -22992.407} C_VEL
LIN {X 0,Y 171.33,Z 329.141,A -85,B 0,C 180,E1 -22997.589,E2 -22997.589} C_VEL
LIN {X 0,Y 171.36,Z 329.119,A -85,B 0,C 180,E1 -23002.034,E2 -23002.034} C_VEL
LIN {X 0,Y 171.393,Z 329.133,A -85,B 0,C 180,E1 -23005.092,E2 -23005.092} C_VEL
LIN {X 0,Y 171.442,Z 329.105,A -85,B 0,C 180,E1 -23010.533,E2 -23010.533} C_VEL
LIN {X 0,Y 171.439,Z 329.127,A -85,B 0,C 180,E1 -23015.799,E2 -23015.799} C_VEL
LIN {X 0,Y 171.572,Z 329.091,A -85,B 0,C 180,E1 -23020.871,E2 -23020.871} C_VEL
LIN {X 0,Y 171.57,Z 329.113,A -85,B 0,C 180,E1 -23025.773,E2 -23025.773} C_VEL
LIN {X 0,Y 171.839,Z 329.053,A -85,B 0,C 180,E1 -23030.585,E2 -23030.585} C_VEL
LIN {X 0,Y 171.803,Z 329.084,A -85,B 0,C 180,E1 -23035.307,E2 -23035.307} C_VEL
LIN {X 0,Y 172.325,Z 328.993,A -85,B 0,C 180,E1 -23040,E2 -23040} C_VEL
LIN {X 0,Y 171.815,Z 329.081,A -85,B 0,C 180,E1 -23044.693,E2 -23044.693} C_VEL
LIN {X 0,Y 171.883,Z 329.055,A -85,B 0,C 180,E1 -23049.414,E2 -23049.414} C_VEL
LIN {X 0,Y 171.573,Z 329.108,A -85,B 0,C 180,E1 -23054.228,E2 -23054.228} C_VEL
LIN {X 0,Y 171.54,Z 329.117,A -85,B 0,C 180,E1 -23059.563,E2 -23059.563} C_VEL
LIN {X 0,Y 171.465,Z 329.124,A -85,B 0,C 180,E1 -23065.618,E2 -23065.618} C_VEL
LIN {X 0,Y 171.438,Z 329.129,A -85,B 0,C 180,E1 -23070.588,E2 -23070.588} C_VEL
LIN {X 0,Y 171.399,Z 329.139,A -85,B 0,C 180,E1 -23075.034,E2 -23075.034} C_VEL
LIN {X 0,Y 171.376,Z 329.143,A -85,B 0,C 180,E1 -23078.818,E2 -23078.818} C_VEL
LIN {X 0,Y 171.318,Z 329.148,A -85,B 0,C 180,E1 -23084.219,E2 -23084.219} C_VEL
LIN {X 0,Y 171.378,Z 329.301,A -85,B 0,C 180,E1 -23085.327,E2 -23085.327} C_VEL
LIN {X 0,Y 172.115,Z 332.015,A -85,B 0,C 180,E1 -23086.997,E2 -23086.997} C_VEL
LIN {X 0,Y 174.414,Z 336.368,A -85,B 0,C 180,E1 -23087.814,E2 -23087.814} C_VEL
LIN {X 0,Y 179.666,Z 346.879,A -85,B 0,C 180,E1 -23089.602,E2 -23089.602} C_VEL
LIN {X 0,Y 184.87,Z 358.804,A -85,B 0,C 180,E1 -23091.308,E2 -23091.308} C_VEL
LIN {X 0,Y 189.461,Z 371.058,A -85,B 0,C 180,E1 -23092.786,E2 -23092.786} C_VEL
LIN {X 0,Y 191.545,Z 393.826,A -85,B 0,C 180,E1 -23094.172,E2 -23094.172} C_VEL
LIN {X 0,Y 189.226,Z 441.512,A -85,B 0,C 180,E1 -23095.883,E2 -23095.883} C_VEL
LIN {X 0,Y 187.86,Z 454.933,A -85,B 0,C 180,E1 -23096.751,E2 -23096.751} C_VEL
LIN {X 0,Y 186.011,Z 467.368,A -85,B 0,C 180,E1 -23097.957,E2 -23097.957} C_VEL
LIN {X 0,Y 184.38,Z 472.771,A -85,B 0,C 180,E1 -23098.516,E2 -23098.516} C_VEL
LIN {X 0,Y 179.927,Z 481.254,A -85,B 0,C 180,E1 -23099.361,E2 -23099.361} C_VEL
LIN {X 0,Y 175.377,Z 489.353,A -85,B 0,C 180,E1 -23100.472,E2 -23100.472} C_VEL
LIN {X 0,Y 173.621,Z 494.145,A -85,B 0,C 180,E1 -23101.44,E2 -23101.44} C_VEL
LIN {X 0,Y 171.142,Z 503.378,A -85,B 0,C 180,E1 -23103.805,E2 -23103.805} C_VEL
LIN {X 0,Y 168.324,Z 513.036,A -85,B 0,C 180,E1 -23106.916,E2 -23106.916} C_VEL
LIN {X 0,Y 166.958,Z 518.34,A -85,B 0,C 180,E1 -23109.036,E2 -23109.036} C_VEL
LIN {X 0,Y 164.815,Z 525.831,A -85,B 0,C 180,E1 -23112.635,E2 -23112.635} C_VEL
LIN {X 0,Y 163.251,Z 531.832,A -85,B 0,C 180,E1 -23116.305,E2 -23116.305} C_VEL
LIN {X 0,Y 162.374,Z 536.565,A -85,B 0,C 180,E1 -23120.032,E2 -23120.032} C_VEL
LIN {X 0,Y 161.974,Z 540.16,A -85,B 0,C 180,E1 -23123.774,E2 -23123.774} C_VEL
LIN {X 0,Y 161.926,Z 542.719,A -85,B 0,C 180,E1 -23127.514,E2 -23127.514} C_VEL
LIN {X 0,Y 162.03,Z 543.909,A -85,B 0,C 180,E1 -23130.001,E2 -23130.001} C_VEL
LIN {X 0,Y 161.834,Z 544.683,A -85,B 0,C 180,E1 -23132.77,E2 -23132.77} C_VEL
LIN {X 0,Y 162.024,Z 544.909,A -85,B 0,C 180,E1 -23137.478,E2 -23137.478} C_VEL
LIN {X 0,Y 162.431,Z 544.477,A -85,B 0,C 180,E1 -23139.968,E2 -23139.968} C_VEL
LIN {X 0,Y 163.096,Z 543.632,A -85,B 0,C 180,E1 -23142.443,E2 -23142.443} C_VEL
LIN {X 0,Y 165.145,Z 540.723,A -85,B 0,C 180,E1 -23147.332,E2 -23147.332} C_VEL
LIN {X 0,Y 167.631,Z 537.436,A -85,B 0,C 180,E1 -23150.878,E2 -23150.878} C_VEL
LIN {X 0,Y 170.681,Z 533.105,A -85,B 0,C 180,E1 -23154.317,E2 -23154.317} C_VEL
LIN {X 0,Y 174.775,Z 526.702,A -85,B 0,C 180,E1 -23158.132,E2 -23158.132} C_VEL
LIN {X 0,Y 179.127,Z 519.485,A -85,B 0,C 180,E1 -23161.324,E2 -23161.324} C_VEL
LIN {X 0,Y 184.07,Z 510.653,A -85,B 0,C 180,E1 -23164.276,E2 -23164.276} C_VEL
LIN {X 0,Y 189.036,Z 500.631,A -85,B 0,C 180,E1 -23166.835,E2 -23166.835} C_VEL
LIN {X 0,Y 193.443,Z 490.397,A -85,B 0,C 180,E1 -23168.809,E2 -23168.809} C_VEL
LIN {X 0,Y 197.433,Z 479.089,A -85,B 0,C 180,E1 -23170.515,E2 -23170.515} C_VEL
LIN {X 0,Y 200.987,Z 467.326,A -85,B 0,C 180,E1 -23171.803,E2 -23171.803} C_VEL
LIN {X 0,Y 203.871,Z 454.41,A -85,B 0,C 180,E1 -23172.826,E2 -23172.826} C_VEL
LIN {X 0,Y 205.812,Z 441.199,A -85,B 0,C 180,E1 -23173.539,E2 -23173.539} C_VEL
LIN {X 0,Y 208.559,Z 403.615,A -85,B 0,C 180,E1 -23174.712,E2 -23174.712} C_VEL
LIN {X 0,Y 207.962,Z 401.297,A -85,B 0,C 180,E1 -23175.022,E2 -23175.022} C_VEL
LIN {X 0,Y 202.437,Z 387.988,A -85,B 0,C 180,E1 -23177.614,E2 -23177.614} C_VEL
LIN {X 0,Y 197.395,Z 377.742,A -85,B 0,C 180,E1 -23180.143,E2 -23180.143} C_VEL
LIN {X 0,Y 192.833,Z 369.41,A -85,B 0,C 180,E1 -23182.641,E2 -23182.641} C_VEL
LIN {X 0,Y 189.618,Z 363.939,A -85,B 0,C 180,E1 -23184.556,E2 -23184.556} C_VEL
LIN {X 0,Y 186.888,Z 359.444,A -85,B 0,C 180,E1 -23186.322,E2 -23186.322} C_VEL
LIN {X 0,Y 183.514,Z 354.172,A -85,B 0,C 180,E1 -23188.708,E2 -23188.708} C_VEL
LIN {X 0,Y 180.438,Z 349.546,A -85,B 0,C 180,E1 -23191.139,E2 -23191.139} C_VEL
LIN {X 0,Y 177.168,Z 345.554,A -85,B 0,C 180,E1 -23194.01,E2 -23194.01} C_VEL
LIN {X 0,Y 175.22,Z 342.579,A -85,B 0,C 180,E1 -23196.039,E2 -23196.039} C_VEL
LIN {X 0,Y 174.728,Z 341.801,A -85,B 0,C 180,E1 -23196.597,E2 -23196.597} C_VEL
LIN {X 0,Y 172.051,Z 339.929,A -85,B 0,C 180,E1 -23199.701,E2 -23199.701} C_VEL
LIN {X 0,Y 170.517,Z 337.137,A -85,B 0,C 180,E1 -23202.149,E2 -23202.149} C_VEL
LIN {X 0,Y 170.152,Z 336.068,A -85,B 0,C 180,E1 -23202.885,E2 -23202.885} C_VEL
LIN {X 0,Y 166.574,Z 333.8,A -85,B 0,C 180,E1 -23212.728,E2 -23212.728} C_VEL
LIN {X 0,Y 166.575,Z 333.521,A -85,B 0,C 180,E1 -23217.582,E2 -23217.582} C_VEL
LIN {X 0,Y 167.127,Z 333.925,A -85,B 0,C 180,E1 -23220.602,E2 -23220.602} C_VEL
LIN {X 0,Y 169.485,Z 335.746,A -85,B 0,C 180,E1 -23226.548,E2 -23226.548} C_VEL
LIN {X 0,Y 170.542,Z 336.279,A -85,B 0,C 180,E1 -23228.287,E2 -23228.287} C_VEL
LIN {X 0,Y 171.563,Z 338.832,A -85,B 0,C 180,E1 -23230.092,E2 -23230.092} C_VEL
LIN {X 0,Y 173.551,Z 341.053,A -85,B 0,C 180,E1 -23232.683,E2 -23232.683} C_VEL
LIN {X 0,Y 175.133,Z 342.112,A -85,B 0,C 180,E1 -23234.377,E2 -23234.377} C_VEL
LIN {X 0,Y 176.99,Z 345.236,A -85,B 0,C 180,E1 -23236.36,E2 -23236.36} C_VEL
LIN {X 0,Y 179.519,Z 347.627,A -85,B 0,C 180,E1 -23238.571,E2 -23238.571} C_VEL
LIN {X 0,Y 181.798,Z 351.006,A -85,B 0,C 180,E1 -23240.471,E2 -23240.471} C_VEL
LIN {X 0,Y 183.576,Z 352.848,A -85,B 0,C 180,E1 -23241.769,E2 -23241.769} C_VEL
LIN {X 0,Y 186.334,Z 356.57,A -85,B 0,C 180,E1 -23243.698,E2 -23243.698} C_VEL
LIN {X 0,Y 190.82,Z 362.74,A -85,B 0,C 180,E1 -23246.505,E2 -23246.505} C_VEL
LIN {X 0,Y 195.935,Z 370.18,A -85,B 0,C 180,E1 -23249.33,E2 -23249.33} C_VEL
LIN {X 0,Y 202.332,Z 380.593,A -85,B 0,C 180,E1 -23252.482,E2 -23252.482} C_VEL
LIN {X 0,Y 206.419,Z 388.056,A -85,B 0,C 180,E1 -23254.326,E2 -23254.326} C_VEL
LIN {X 0,Y 209.078,Z 393.85,A -85,B 0,C 180,E1 -23255.501,E2 -23255.501} C_VEL
LIN {X 0,Y 206.476,Z 430.14,A -85,B 0,C 180,E1 -23256.632,E2 -23256.632} C_VEL
LIN {X 0,Y 204.594,Z 443.765,A -85,B 0,C 180,E1 -23257.39,E2 -23257.39} C_VEL
LIN {X 0,Y 202.383,Z 454.292,A -85,B 0,C 180,E1 -23258.217,E2 -23258.217} C_VEL
LIN {X 0,Y 199.29,Z 466.659,A -85,B 0,C 180,E1 -23259.621,E2 -23259.621} C_VEL
LIN {X 0,Y 195.885,Z 476.915,A -85,B 0,C 180,E1 -23261.11,E2 -23261.11} C_VEL
LIN {X 0,Y 191.652,Z 487.863,A -85,B 0,C 180,E1 -23263.211,E2 -23263.211} C_VEL
LIN {X 0,Y 187.283,Z 497.22,A -85,B 0,C 180,E1 -23265.479,E2 -23265.479} C_VEL
LIN {X 0,Y 183.246,Z 504.878,A -85,B 0,C 180,E1 -23267.841,E2 -23267.841} C_VEL
LIN {X 0,Y 178.614,Z 512.79,A -85,B 0,C 180,E1 -23270.982,E2 -23270.982} C_VEL
LIN {X 0,Y 174.493,Z 519.068,A -85,B 0,C 180,E1 -23274.266,E2 -23274.266} C_VEL
LIN {X 0,Y 170.946,Z 524.018,A -85,B 0,C 180,E1 -23277.692,E2 -23277.692} C_VEL
LIN {X 0,Y 167.77,Z 528.117,A -85,B 0,C 180,E1 -23281.607,E2 -23281.607} C_VEL
LIN {X 0,Y 165.664,Z 530.515,A -85,B 0,C 180,E1 -23284.897,E2 -23284.897} C_VEL
LIN {X 0,Y 164.401,Z 531.778,A -85,B 0,C 180,E1 -23287.371,E2 -23287.371} C_VEL
LIN {X 0,Y 162.911,Z 532.961,A -85,B 0,C 180,E1 -23291.637,E2 -23291.637} C_VEL
LIN {X 0,Y 162.195,Z 533.044,A -85,B 0,C 180,E1 -23294.93,E2 -23294.93} C_VEL
LIN {X 0,Y 161.814,Z 532.665,A -85,B 0,C 180,E1 -23297.456,E2 -23297.456} C_VEL
LIN {X 0,Y 161.718,Z 531.885,A -85,B 0,C 180,E1 -23299.988,E2 -23299.988} C_VEL
LIN {X 0,Y 161.802,Z 530.66,A -85,B 0,C 180,E1 -23302.511,E2 -23302.511} C_VEL
LIN {X 0,Y 162.159,Z 528.735,A -85,B 0,C 180,E1 -23305.43,E2 -23305.43} C_VEL
LIN {X 0,Y 162.67,Z 525.783,A -85,B 0,C 180,E1 -23308.761,E2 -23308.761} C_VEL
LIN {X 0,Y 163.616,Z 521.483,A -85,B 0,C 180,E1 -23312.461,E2 -23312.461} C_VEL
LIN {X 0,Y 165.105,Z 515.997,A -85,B 0,C 180,E1 -23316.107,E2 -23316.107} C_VEL
LIN {X 0,Y 167.085,Z 509.156,A -85,B 0,C 180,E1 -23319.685,E2 -23319.685} C_VEL
LIN {X 0,Y 169.641,Z 500.599,A -85,B 0,C 180,E1 -23323.169,E2 -23323.169} C_VEL
LIN {X 0,Y 172.155,Z 491.821,A -85,B 0,C 180,E1 -23325.994,E2 -23325.994} C_VEL
LIN {X 0,Y 175.101,Z 481.004,A -85,B 0,C 180,E1 -23328.728,E2 -23328.728} C_VEL
LIN {X 0,Y 177.74,Z 470.098,A -85,B 0,C 180,E1 -23330.845,E2 -23330.845} C_VEL
LIN {X 0,Y 179.811,Z 459.874,A -85,B 0,C 180,E1 -23332.399,E2 -23332.399} C_VEL
LIN {X 0,Y 181.636,Z 446.502,A -85,B 0,C 180,E1 -23333.969,E2 -23333.969} C_VEL
LIN {X 0,Y 182.828,Z 436.305,A -85,B 0,C 180,E1 -23334.785,E2 -23334.785} C_VEL
LIN {X 0,Y 183.892,Z 423.527,A -85,B 0,C 180,E1 -23335.434,E2 -23335.434} C_VEL
LIN {X 0,Y 186.419,Z 371.924,A -85,B 0,C 180,E1 -23337.274,E2 -23337.274} C_VEL
LIN {X 0,Y 183.543,Z 364.837,A -85,B 0,C 180,E1 -23338.192,E2 -23338.192} C_VEL
LIN {X 0,Y 176.833,Z 351.469,A -85,B 0,C 180,E1 -23340.332,E2 -23340.332} C_VEL
LIN {X 0,Y 170.362,Z 340.447,A -85,B 0,C 180,E1 -23342.519,E2 -23342.519} C_VEL
LIN {X 0,Y 168.262,Z 337.138,A -85,B 0,C 180,E1 -23343.266,E2 -23343.266} C_VEL
LIN {X 0,Y 166.506,Z 334.246,A -85,B 0,C 180,E1 -23343.917,E2 -23343.917} C_VEL
LIN {X 0,Y 164.843,Z 331.846,A -85,B 0,C 180,E1 -23344.534,E2 -23344.534} C_VEL
LIN {X 0,Y 164.367,Z 330.009,A -85,B 0,C 180,E1 -23344.827,E2 -23344.827} C_VEL
LIN {X 0,Y 164.282,Z 330.016,A -85,B 0,C 180,E1 -23349.916,E2 -23349.916} C_VEL
LIN {X 0,Y 164.276,Z 330.007,A -85,B 0,C 180,E1 -23353.341,E2 -23353.341} C_VEL
LIN {X 0,Y 164.258,Z 330.02,A -85,B 0,C 180,E1 -23356.798,E2 -23356.798} C_VEL
LIN {X 0,Y 164.287,Z 330.001,A -85,B 0,C 180,E1 -23360.352,E2 -23360.352} C_VEL
LIN {X 0,Y 164.321,Z 330.013,A -85,B 0,C 180,E1 -23366.22,E2 -23366.22} C_VEL
LIN {X 0,Y 164.384,Z 329.984,A -85,B 0,C 180,E1 -23369.134,E2 -23369.134} C_VEL
LIN {X 0,Y 164.401,Z 330.006,A -85,B 0,C 180,E1 -23374.692,E2 -23374.692} C_VEL
LIN {X 0,Y 164.479,Z 329.969,A -85,B 0,C 180,E1 -23380.051,E2 -23380.051} C_VEL
LIN {X 0,Y 164.518,Z 329.991,A -85,B 0,C 180,E1 -23385.149,E2 -23385.149} C_VEL
LIN {X 0,Y 164.76,Z 329.933,A -85,B 0,C 180,E1 -23390.176,E2 -23390.176} C_VEL
LIN {X 0,Y 164.82,Z 329.941,A -85,B 0,C 180,E1 -23392.651,E2 -23392.651} C_VEL
LIN {X 0,Y 165.039,Z 329.919,A -85,B 0,C 180,E1 -23397.56,E2 -23397.56} C_VEL
LIN {X 0,Y 165.287,Z 329.868,A -85,B 0,C 180,E1 -23400,E2 -23400} C_VEL
LIN {X 0,Y 164.765,Z 329.961,A -85,B 0,C 180,E1 -23404.894,E2 -23404.894} C_VEL
LIN {X 0,Y 164.845,Z 329.948,A -85,B 0,C 180,E1 -23407.349,E2 -23407.349} C_VEL
LIN {X 0,Y 164.737,Z 329.937,A -85,B 0,C 180,E1 -23411.132,E2 -23411.132} C_VEL
LIN {X 0,Y 164.478,Z 329.992,A -85,B 0,C 180,E1 -23417.404,E2 -23417.404} C_VEL
LIN {X 0,Y 164.469,Z 329.998,A -85,B 0,C 180,E1 -23419.99,E2 -23419.99} C_VEL
LIN {X 0,Y 164.39,Z 330.004,A -85,B 0,C 180,E1 -23426.135,E2 -23426.135} C_VEL
LIN {X 0,Y 164.372,Z 330.012,A -85,B 0,C 180,E1 -23431.229,E2 -23431.229} C_VEL
LIN {X 0,Y 164.308,Z 330.019,A -85,B 0,C 180,E1 -23436.786,E2 -23436.786} C_VEL
LIN {X 0,Y 164.296,Z 330.021,A -85,B 0,C 180,E1 -23439.915,E2 -23439.915} C_VEL
LIN {X 0,Y 164.301,Z 330.107,A -85,B 0,C 180,E1 -23443.917,E2 -23443.917} C_VEL
LIN {X 0,Y 164.774,Z 331.785,A -85,B 0,C 180,E1 -23444.944,E2 -23444.944} C_VEL
LIN {X 0,Y 166.951,Z 335.791,A -85,B 0,C 180,E1 -23445.794,E2 -23445.794} C_VEL
LIN {X 0,Y 173.828,Z 348.9,A -85,B 0,C 180,E1 -23448.306,E2 -23448.306} C_VEL
LIN {X 0,Y 179.745,Z 362.826,A -85,B 0,C 180,E1 -23450.389,E2 -23450.389} C_VEL
LIN {X 0,Y 183.655,Z 373.422,A -85,B 0,C 180,E1 -23451.73,E2 -23451.73} C_VEL
LIN {X 0,Y 185.49,Z 394.099,A -85,B 0,C 180,E1 -23453.044,E2 -23453.044} C_VEL
LIN {X 0,Y 183.115,Z 441.207,A -85,B 0,C 180,E1 -23454.78,E2 -23454.78} C_VEL
LIN {X 0,Y 181.63,Z 455.098,A -85,B 0,C 180,E1 -23455.705,E2 -23455.705} C_VEL
LIN {X 0,Y 179.661,Z 467.621,A -85,B 0,C 180,E1 -23456.963,E2 -23456.963} C_VEL
LIN {X 0,Y 177.213,Z 479.57,A -85,B 0,C 180,E1 -23458.635,E2 -23458.635} C_VEL
LIN {X 0,Y 174.385,Z 491.04,A -85,B 0,C 180,E1 -23460.749,E2 -23460.749} C_VEL
LIN {X 0,Y 173.621,Z 494.145,A -85,B 0,C 180,E1 -23461.44,E2 -23461.44} C_VEL
LIN {X 0,Y 171.868,Z 498.828,A -85,B 0,C 180,E1 -23462.5,E2 -23462.5} C_VEL
LIN {X 0,Y 167.219,Z 505.984,A -85,B 0,C 180,E1 -23464.186,E2 -23464.186} C_VEL
LIN {X 0,Y 162.5,Z 512.651,A -85,B 0,C 180,E1 -23466.146,E2 -23466.146} C_VEL
LIN {X 0,Y 160.687,Z 516.465,A -85,B 0,C 180,E1 -23467.612,E2 -23467.612} C_VEL
LIN {X 0,Y 158.357,Z 524.092,A -85,B 0,C 180,E1 -23471.232,E2 -23471.232} C_VEL
LIN {X 0,Y 156.302,Z 531.286,A -85,B 0,C 180,E1 -23475.684,E2 -23475.684} C_VEL
LIN {X 0,Y 155.338,Z 536.08,A -85,B 0,C 180,E1 -23479.575,E2 -23479.575} C_VEL
LIN {X 0,Y 154.899,Z 539.732,A -85,B 0,C 180,E1 -23483.488,E2 -23483.488} C_VEL
LIN {X 0,Y 154.845,Z 542.344,A -85,B 0,C 180,E1 -23487.4,E2 -23487.4} C_VEL
LIN {X 0,Y 154.936,Z 543.562,A -85,B 0,C 180,E1 -23490.001,E2 -23490.001} C_VEL
LIN {X 0,Y 154.777,Z 544.333,A -85,B 0,C 180,E1 -23492.604,E2 -23492.604} C_VEL
LIN {X 0,Y 154.97,Z 544.656,A -85,B 0,C 180,E1 -23497.821,E2 -23497.821} C_VEL
LIN {X 0,Y 156.122,Z 543.449,A -85,B 0,C 180,E1 -23503.009,E2 -23503.009} C_VEL
LIN {X 0,Y 158.369,Z 540.593,A -85,B 0,C 180,E1 -23508.099,E2 -23508.099} C_VEL
LIN {X 0,Y 161.001,Z 537.36,A -85,B 0,C 180,E1 -23511.781,E2 -23511.781} C_VEL
LIN {X 0,Y 165.039,Z 531.954,A -85,B 0,C 180,E1 -23516.15,E2 -23516.15} C_VEL
LIN {X 0,Y 169.294,Z 525.573,A -85,B 0,C 180,E1 -23519.88,E2 -23519.88} C_VEL
LIN {X 0,Y 173.936,Z 518.286,A -85,B 0,C 180,E1 -23523.058,E2 -23523.058} C_VEL
LIN {X 0,Y 179.18,Z 509.27,A -85,B 0,C 180,E1 -23526.041,E2 -23526.041} C_VEL
LIN {X 0,Y 183.893,Z 499.973,A -85,B 0,C 180,E1 -23528.393,E2 -23528.393} C_VEL
LIN {X 0,Y 188.479,Z 489.653,A -85,B 0,C 180,E1 -23530.383,E2 -23530.383} C_VEL
LIN {X 0,Y 192.117,Z 479.809,A -85,B 0,C 180,E1 -23531.884,E2 -23531.884} C_VEL
LIN {X 0,Y 196.067,Z 467.309,A -85,B 0,C 180,E1 -23533.278,E2 -23533.278} C_VEL
LIN {X 0,Y 199.04,Z 454.525,A -85,B 0,C 180,E1 -23534.305,E2 -23534.305} C_VEL
LIN {X 0,Y 201.116,Z 441.028,A -85,B 0,C 180,E1 -23535.039,E2 -23535.039} C_VEL
LIN {X 0,Y 203.796,Z 405.245,A -85,B 0,C 180,E1 -23536.182,E2 -23536.182} C_VEL
LIN {X 0,Y 198.576,Z 392.251,A -85,B 0,C 180,E1 -23538.8,E2 -23538.8} C_VEL
LIN {X 0,Y 193.385,Z 381.494,A -85,B 0,C 180,E1 -23541.594,E2 -23541.594} C_VEL
LIN {X 0,Y 189.271,Z 373.862,A -85,B 0,C 180,E1 -23544.017,E2 -23544.017} C_VEL
LIN {X 0,Y 184.985,Z 366.208,A -85,B 0,C 180,E1 -23546.849,E2 -23546.849} C_VEL
LIN {X 0,Y 181.124,Z 360.105,A -85,B 0,C 180,E1 -23549.706,E2 -23549.706} C_VEL
LIN {X 0,Y 177.768,Z 354.906,A -85,B 0,C 180,E1 -23552.559,E2 -23552.559} C_VEL
LIN {X 0,Y 173.716,Z 349.477,A -85,B 0,C 180,E1 -23556.61,E2 -23556.61} C_VEL
LIN {X 0,Y 173.25,Z 348.609,A -85,B 0,C 180,E1 -23557.175,E2 -23557.175} C_VEL
LIN {X 0,Y 170.639,Z 346.589,A -85,B 0,C 180,E1 -23560.371,E2 -23560.371} C_VEL
LIN {X 0,Y 169.137,Z 343.703,A -85,B 0,C 180,E1 -23562.947,E2 -23562.947} C_VEL
LIN {X 0,Y 168.941,Z 343.061,A -85,B 0,C 180,E1 -23563.381,E2 -23563.381} C_VEL
LIN {X 0,Y 165.708,Z 340.846,A -85,B 0,C 180,E1 -23572.69,E2 -23572.69} C_VEL
LIN {X 0,Y 165.877,Z 340.654,A -85,B 0,C 180,E1 -23578.786,E2 -23578.786} C_VEL
LIN {X 0,Y 166.855,Z 341.752,A -85,B 0,C 180,E1 -23582.716,E2 -23582.716} C_VEL
LIN {X 0,Y 169.199,Z 343.081,A -85,B 0,C 180,E1 -23587.581,E2 -23587.581} C_VEL
LIN {X 0,Y 170.676,Z 346.305,A -85,B 0,C 180,E1 -23590.187,E2 -23590.187} C_VEL
LIN {X 0,Y 173.097,Z 348.428,A -85,B 0,C 180,E1 -23593.202,E2 -23593.202} C_VEL
LIN {X 0,Y 173.76,Z 349.353,A -85,B 0,C 180,E1 -23593.97,E2 -23593.97} C_VEL
LIN {X 0,Y 176.109,Z 352.676,A -85,B 0,C 180,E1 -23596.445,E2 -23596.445} C_VEL
LIN {X 0,Y 177.6,Z 354.112,A -85,B 0,C 180,E1 -23597.785,E2 -23597.785} C_VEL
LIN {X 0,Y 180.123,Z 357.726,A -85,B 0,C 180,E1 -23599.962,E2 -23599.962} C_VEL
LIN {X 0,Y 181.507,Z 359.302,A -85,B 0,C 180,E1 -23601.024,E2 -23601.024} C_VEL
LIN {X 0,Y 184.376,Z 363.12,A -85,B 0,C 180,E1 -23603.106,E2 -23603.106} C_VEL
LIN {X 0,Y 190.242,Z 371.629,A -85,B 0,C 180,E1 -23606.851,E2 -23606.851} C_VEL
LIN {X 0,Y 195.08,Z 379.261,A -85,B 0,C 180,E1 -23609.545,E2 -23609.545} C_VEL
LIN {X 0,Y 200.415,Z 388.445,A -85,B 0,C 180,E1 -23612.226,E2 -23612.226} C_VEL
LIN {X 0,Y 203.789,Z 395.271,A -85,B 0,C 180,E1 -23613.823,E2 -23613.823} C_VEL
LIN {X 0,Y 204.285,Z 396.456,A -85,B 0,C 180,E1 -23614.059,E2 -23614.059} C_VEL
LIN {X 0,Y 201.689,Z 431.29,A -85,B 0,C 180,E1 -23615.183,E2 -23615.183} C_VEL
LIN {X 0,Y 199.693,Z 444.826,A -85,B 0,C 180,E1 -23615.956,E2 -23615.956} C_VEL
LIN {X 0,Y 197.435,Z 455.075,A -85,B 0,C 180,E1 -23616.783,E2 -23616.783} C_VEL
LIN {X 0,Y 194.655,Z 465.86,A -85,B 0,C 180,E1 -23618.018,E2 -23618.018} C_VEL
LIN {X 0,Y 191.158,Z 476.092,A -85,B 0,C 180,E1 -23619.459,E2 -23619.459} C_VEL
LIN {X 0,Y 187.221,Z 486.187,A -85,B 0,C 180,E1 -23621.342,E2 -23621.342} C_VEL
LIN {X 0,Y 182.563,Z 496.096,A -85,B 0,C 180,E1 -23623.702,E2 -23623.702} C_VEL
LIN {X 0,Y 177.928,Z 504.556,A -85,B 0,C 180,E1 -23626.271,E2 -23626.271} C_VEL
LIN {X 0,Y 173.008,Z 512.605,A -85,B 0,C 180,E1 -23629.461,E2 -23629.461} C_VEL
LIN {X 0,Y 168.533,Z 519.116,A -85,B 0,C 180,E1 -23632.909,E2 -23632.909} C_VEL
LIN {X 0,Y 164.839,Z 524.001,A -85,B 0,C 180,E1 -23636.339,E2 -23636.339} C_VEL
LIN {X 0,Y 161.08,Z 528.507,A -85,B 0,C 180,E1 -23640.763,E2 -23640.763} C_VEL
LIN {X 0,Y 159.08,Z 530.638,A -85,B 0,C 180,E1 -23643.781,E2 -23643.781} C_VEL
LIN {X 0,Y 157.717,Z 531.934,A -85,B 0,C 180,E1 -23646.355,E2 -23646.355} C_VEL
LIN {X 0,Y 155.904,Z 533.253,A -85,B 0,C 180,E1 -23651.201,E2 -23651.201} C_VEL
LIN {X 0,Y 155.203,Z 533.33,A -85,B 0,C 180,E1 -23654.234,E2 -23654.234} C_VEL
LIN {X 0,Y 154.616,Z 532.243,A -85,B 0,C 180,E1 -23659.523,E2 -23659.523} C_VEL
LIN {X 0,Y 154.688,Z 531.072,A -85,B 0,C 180,E1 -23662.165,E2 -23662.165} C_VEL
LIN {X 0,Y 155.082,Z 528.949,A -85,B 0,C 180,E1 -23665.553,E2 -23665.553} C_VEL
LIN {X 0,Y 155.783,Z 525.034,A -85,B 0,C 180,E1 -23669.999,E2 -23669.999} C_VEL
LIN {X 0,Y 156.991,Z 520.423,A -85,B 0,C 180,E1 -23673.849,E2 -23673.849} C_VEL
LIN {X 0,Y 158.983,Z 513.468,A -85,B 0,C 180,E1 -23678.259,E2 -23678.259} C_VEL
LIN {X 0,Y 161.351,Z 505.944,A -85,B 0,C 180,E1 -23681.939,E2 -23681.939} C_VEL
LIN {X 0,Y 163.725,Z 498.261,A -85,B 0,C 180,E1 -23684.923,E2 -23684.923} C_VEL
LIN {X 0,Y 166.831,Z 487.817,A -85,B 0,C 180,E1 -23688.099,E2 -23688.099} C_VEL
LIN {X 0,Y 169.699,Z 477.182,A -85,B 0,C 180,E1 -23690.609,E2 -23690.609} C_VEL
LIN {X 0,Y 172.299,Z 466.859,A -85,B 0,C 180,E1 -23692.481,E2 -23692.481} C_VEL
LIN {X 0,Y 174.466,Z 454.639,A -85,B 0,C 180,E1 -23694.227,E2 -23694.227} C_VEL
LIN {X 0,Y 176.157,Z 441.101,A -85,B 0,C 180,E1 -23695.633,E2 -23695.633} C_VEL
LIN {X 0,Y 177.551,Z 428.258,A -85,B 0,C 180,E1 -23696.425,E2 -23696.425} C_VEL
LIN {X 0,Y 180.438,Z 373.749,A -85,B 0,C 180,E1 -23698.437,E2 -23698.437} C_VEL
LIN {X 0,Y 175.815,Z 363.299,A -85,B 0,C 180,E1 -23699.986,E2 -23699.986} C_VEL
LIN {X 0,Y 169.557,Z 351.362,A -85,B 0,C 180,E1 -23702.155,E2 -23702.155} C_VEL
LIN {X 0,Y 164.115,Z 342.246,A -85,B 0,C 180,E1 -23704.163,E2 -23704.163} C_VEL
LIN {X 0,Y 161.348,Z 338.143,A -85,B 0,C 180,E1 -23705.226,E2 -23705.226} C_VEL
LIN {X 0,Y 159.678,Z 335.371,A -85,B 0,C 180,E1 -23705.912,E2 -23705.912} C_VEL
LIN {X 0,Y 157.852,Z 333.012,A -85,B 0,C 180,E1 -23706.646,E2 -23706.646} C_VEL
LIN {X 0,Y 157.217,Z 330.895,A -85,B 0,C 180,E1 -23707.07,E2 -23707.07} C_VEL
LIN {X 0,Y 157.185,Z 330.9,A -85,B 0,C 180,E1 -23712.116,E2 -23712.116} C_VEL
LIN {X 0,Y 157.187,Z 330.902,A -85,B 0,C 180,E1 -23717.882,E2 -23717.882} C_VEL
LIN {X 0,Y 157.256,Z 330.885,A -85,B 0,C 180,E1 -23723.554,E2 -23723.554} C_VEL
LIN {X 0,Y 157.288,Z 330.874,A -85,B 0,C 180,E1 -23728.096,E2 -23728.096} C_VEL
LIN {X 0,Y 157.309,Z 330.886,A -85,B 0,C 180,E1 -23733.464,E2 -23733.464} C_VEL
LIN {X 0,Y 157.386,Z 330.851,A -85,B 0,C 180,E1 -23739.67,E2 -23739.67} C_VEL
LIN {X 0,Y 157.448,Z 330.873,A -85,B 0,C 180,E1 -23744.466,E2 -23744.466} C_VEL
LIN {X 0,Y 157.682,Z 330.813,A -85,B 0,C 180,E1 -23749.731,E2 -23749.731} C_VEL
LIN {X 0,Y 157.757,Z 330.817,A -85,B 0,C 180,E1 -23752.32,E2 -23752.32} C_VEL
LIN {X 0,Y 158.25,Z 330.743,A -85,B 0,C 180,E1 -23760,E2 -23760} C_VEL
LIN {X 0,Y 157.802,Z 330.822,A -85,B 0,C 180,E1 -23767.679,E2 -23767.679} C_VEL
LIN {X 0,Y 157.667,Z 330.817,A -85,B 0,C 180,E1 -23771.302,E2 -23771.302} C_VEL
LIN {X 0,Y 157.449,Z 330.872,A -85,B 0,C 180,E1 -23775.535,E2 -23775.535} C_VEL
LIN {X 0,Y 157.366,Z 330.882,A -85,B 0,C 180,E1 -23780.934,E2 -23780.934} C_VEL
LIN {X 0,Y 157.311,Z 330.887,A -85,B 0,C 180,E1 -23786.686,E2 -23786.686} C_VEL
LIN {X 0,Y 157.274,Z 330.898,A -85,B 0,C 180,E1 -23792.428,E2 -23792.428} C_VEL
LIN {X 0,Y 157.278,Z 330.895,A -85,B 0,C 180,E1 -23796.457,E2 -23796.457} C_VEL
LIN {X 0,Y 157.242,Z 331.104,A -85,B 0,C 180,E1 -23802.486,E2 -23802.486} C_VEL
LIN {X 0,Y 158.445,Z 334.066,A -85,B 0,C 180,E1 -23803.113,E2 -23803.113} C_VEL
LIN {X 0,Y 160.622,Z 337.108,A -85,B 0,C 180,E1 -23803.989,E2 -23803.989} C_VEL
LIN {X 0,Y 167.609,Z 350.318,A -85,B 0,C 180,E1 -23806.766,E2 -23806.766} C_VEL
LIN {X 0,Y 173.088,Z 362.742,A -85,B 0,C 180,E1 -23808.829,E2 -23808.829} C_VEL
LIN {X 0,Y 177.877,Z 375.626,A -85,B 0,C 180,E1 -23810.589,E2 -23810.589} C_VEL
LIN {X 0,Y 179.467,Z 395.535,A -85,B 0,C 180,E1 -23811.886,E2 -23811.886} C_VEL
LIN {X 0,Y 177.022,Z 441.437,A -85,B 0,C 180,E1 -23813.629,E2 -23813.629} C_VEL
LIN {X 0,Y 175.47,Z 455.264,A -85,B 0,C 180,E1 -23814.586,E2 -23814.586} C_VEL
LIN {X 0,Y 173.523,Z 467.121,A -85,B 0,C 180,E1 -23815.81,E2 -23815.81} C_VEL
LIN {X 0,Y 171.15,Z 478.331,A -85,B 0,C 180,E1 -23817.389,E2 -23817.389} C_VEL
LIN {X 0,Y 168.235,Z 489.988,A -85,B 0,C 180,E1 -23819.57,E2 -23819.57} C_VEL
LIN {X 0,Y 165.358,Z 500.49,A -85,B 0,C 180,E1 -23822.129,E2 -23822.129} C_VEL
LIN {X 0,Y 162.612,Z 509.747,A -85,B 0,C 180,E1 -23825.012,E2 -23825.012} C_VEL
LIN {X 0,Y 160.687,Z 516.465,A -85,B 0,C 180,E1 -23827.612,E2 -23827.612} C_VEL
LIN {X 0,Y 158.935,Z 520.109,A -85,B 0,C 180,E1 -23829.171,E2 -23829.171} C_VEL
LIN {X 0,Y 154.476,Z 525.445,A -85,B 0,C 180,E1 -23831.748,E2 -23831.748} C_VEL
LIN {X 0,Y 150.246,Z 530.192,A -85,B 0,C 180,E1 -23834.618,E2 -23834.618} C_VEL
LIN {X 0,Y 148.906,Z 532.782,A -85,B 0,C 180,E1 -23836.589,E2 -23836.589} C_VEL
LIN {X 0,Y 148.122,Z 536.959,A -85,B 0,C 180,E1 -23840.442,E2 -23840.442} C_VEL
LIN {X 0,Y 147.756,Z 540.311,A -85,B 0,C 180,E1 -23844.543,E2 -23844.543} C_VEL
LIN {X 0,Y 147.756,Z 541.969,A -85,B 0,C 180,E1 -23847.275,E2 -23847.275} C_VEL
LIN {X 0,Y 147.844,Z 543.212,A -85,B 0,C 180,E1 -23850.001,E2 -23850.001} C_VEL
LIN {X 0,Y 147.678,Z 544.027,A -85,B 0,C 180,E1 -23852.729,E2 -23852.729} C_VEL
LIN {X 0,Y 147.938,Z 544.403,A -85,B 0,C 180,E1 -23858.195,E2 -23858.195} C_VEL
LIN {X 0,Y 149.17,Z 543.255,A -85,B 0,C 180,E1 -23863.627,E2 -23863.627} C_VEL
LIN {X 0,Y 150.189,Z 542.064,A -85,B 0,C 180,E1 -23866.307,E2 -23866.307} C_VEL
LIN {X 0,Y 153.425,Z 538.463,A -85,B 0,C 180,E1 -23871.499,E2 -23871.499} C_VEL
LIN {X 0,Y 156.597,Z 534.599,A -85,B 0,C 180,E1 -23875.238,E2 -23875.238} C_VEL
LIN {X 0,Y 160.344,Z 529.635,A -85,B 0,C 180,E1 -23878.826,E2 -23878.826} C_VEL
LIN {X 0,Y 164.707,Z 523.422,A -85,B 0,C 180,E1 -23882.234,E2 -23882.234} C_VEL
LIN {X 0,Y 169.815,Z 515.699,A -85,B 0,C 180,E1 -23885.41,E2 -23885.41} C_VEL
LIN {X 0,Y 175.416,Z 506.05,A -85,B 0,C 180,E1 -23888.39,E2 -23888.39} C_VEL
LIN {X 0,Y 180.483,Z 496.108,A -85,B 0,C 180,E1 -23890.712,E2 -23890.712} C_VEL
LIN {X 0,Y 185.324,Z 484.893,A -85,B 0,C 180,E1 -23892.678,E2 -23892.678} C_VEL
LIN {X 0,Y 188.65,Z 475.692,A -85,B 0,C 180,E1 -23893.937,E2 -23893.937} C_VEL
LIN {X 0,Y 192.44,Z 462.921,A -85,B 0,C 180,E1 -23895.225,E2 -23895.225} C_VEL
LIN {X 0,Y 195.198,Z 450.206,A -85,B 0,C 180,E1 -23896.14,E2 -23896.14} C_VEL
LIN {X 0,Y 196.972,Z 437.19,A -85,B 0,C 180,E1 -23896.747,E2 -23896.747} C_VEL
LIN {X 0,Y 199.203,Z 407.806,A -85,B 0,C 180,E1 -23897.657,E2 -23897.657} C_VEL
LIN {X 0,Y 194.438,Z 395.712,A -85,B 0,C 180,E1 -23900.237,E2 -23900.237} C_VEL
LIN {X 0,Y 189.35,Z 384.907,A -85,B 0,C 180,E1 -23903.202,E2 -23903.202} C_VEL
LIN {X 0,Y 184.268,Z 375.425,A -85,B 0,C 180,E1 -23906.521,E2 -23906.521} C_VEL
LIN {X 0,Y 181.327,Z 370.278,A -85,B 0,C 180,E1 -23908.682,E2 -23908.682} C_VEL
LIN {X 0,Y 178.948,Z 366.278,A -85,B 0,C 180,E1 -23910.598,E2 -23910.598} C_VEL
LIN {X 0,Y 175.803,Z 361.223,A -85,B 0,C 180,E1 -23913.433,E2 -23913.433} C_VEL
LIN {X 0,Y 172.013,Z 355.854,A -85,B 0,C 180,E1 -23917.478,E2 -23917.478} C_VEL
LIN {X 0,Y 170.472,Z 354.567,A -85,B 0,C 180,E1 -23919.329,E2 -23919.329} C_VEL
LIN {X 0,Y 168.373,Z 351.773,A -85,B 0,C 180,E1 -23922.555,E2 -23922.555} C_VEL
LIN {X 0,Y 167.657,Z 349.976,A -85,B 0,C 180,E1 -23924.059,E2 -23924.059} C_VEL
LIN {X 0,Y 164.842,Z 347.905,A -85,B 0,C 180,E1 -23932.651,E2 -23932.651} C_VEL
LIN {X 0,Y 165.005,Z 347.703,A -85,B 0,C 180,E1 -23938.779,E2 -23938.779} C_VEL
LIN {X 0,Y 165.879,Z 348.722,A -85,B 0,C 180,E1 -23942.428,E2 -23942.428} C_VEL
LIN {X 0,Y 167.998,Z 350.154,A -85,B 0,C 180,E1 -23947.096,E2 -23947.096} C_VEL
LIN {X 0,Y 169.889,Z 353.745,A -85,B 0,C 180,E1 -23950.393,E2 -23950.393} C_VEL
LIN {X 0,Y 172.02,Z 355.66,A -85,B 0,C 180,E1 -23953.06,E2 -23953.06} C_VEL
LIN {X 0,Y 174.448,Z 359.281,A -85,B 0,C 180,E1 -23955.779,E2 -23955.779} C_VEL
LIN {X 0,Y 175.843,Z 360.759,A -85,B 0,C 180,E1 -23957.104,E2 -23957.104} C_VEL
LIN {X 0,Y 178.474,Z 364.453,A -85,B 0,C 180,E1 -23959.453,E2 -23959.453} C_VEL
LIN {X 0,Y 179.975,Z 366.563,A -85,B 0,C 180,E1 -23960.674,E2 -23960.674} C_VEL
LIN {X 0,Y 182.72,Z 370.328,A -85,B 0,C 180,E1 -23962.724,E2 -23962.724} C_VEL
LIN {X 0,Y 187.404,Z 377.231,A -85,B 0,C 180,E1 -23965.846,E2 -23965.846} C_VEL
LIN {X 0,Y 192.345,Z 385.283,A -85,B 0,C 180,E1 -23968.75,E2 -23968.75} C_VEL
LIN {X 0,Y 197.332,Z 394.262,A -85,B 0,C 180,E1 -23971.391,E2 -23971.391} C_VEL
LIN {X 0,Y 199.68,Z 399.16,A -85,B 0,C 180,E1 -23972.574,E2 -23972.574} C_VEL
LIN {X 0,Y 197.101,Z 431.795,A -85,B 0,C 180,E1 -23973.63,E2 -23973.63} C_VEL
LIN {X 0,Y 195.087,Z 445.004,A -85,B 0,C 180,E1 -23974.391,E2 -23974.391} C_VEL
LIN {X 0,Y 192.617,Z 455.846,A -85,B 0,C 180,E1 -23975.274,E2 -23975.274} C_VEL
LIN {X 0,Y 189.345,Z 467.626,A -85,B 0,C 180,E1 -23976.65,E2 -23976.65} C_VEL
LIN {X 0,Y 185.575,Z 478.029,A -85,B 0,C 180,E1 -23978.201,E2 -23978.201} C_VEL
LIN {X 0,Y 180.982,Z 488.876,A -85,B 0,C 180,E1 -23980.35,E2 -23980.35} C_VEL
LIN {X 0,Y 176.302,Z 498.065,A -85,B 0,C 180,E1 -23982.662,E2 -23982.662} C_VEL
LIN {X 0,Y 171.834,Z 505.743,A -85,B 0,C 180,E1 -23985.127,E2 -23985.127} C_VEL
LIN {X 0,Y 166.711,Z 513.57,A -85,B 0,C 180,E1 -23988.396,E2 -23988.396} C_VEL
LIN {X 0,Y 162.582,Z 519.258,A -85,B 0,C 180,E1 -23991.508,E2 -23991.508} C_VEL
LIN {X 0,Y 158.818,Z 523.988,A -85,B 0,C 180,E1 -23994.88,E2 -23994.88} C_VEL
LIN {X 0,Y 155.27,Z 528.018,A -85,B 0,C 180,E1 -23998.783,E2 -23998.783} C_VEL
LIN {X 0,Y 152.579,Z 530.764,A -85,B 0,C 180,E1 -24002.572,E2 -24002.572} C_VEL
LIN {X 0,Y 151.055,Z 532.092,A -85,B 0,C 180,E1 -24005.244,E2 -24005.244} C_VEL
LIN {X 0,Y 149.85,Z 533.016,A -85,B 0,C 180,E1 -24007.962,E2 -24007.962} C_VEL
LIN {X 0,Y 148.921,Z 533.538,A -85,B 0,C 180,E1 -24010.709,E2 -24010.709} C_VEL
LIN {X 0,Y 148.23,Z 533.616,A -85,B 0,C 180,E1 -24013.471,E2 -24013.471} C_VEL
LIN {X 0,Y 147.535,Z 532.591,A -85,B 0,C 180,E1 -24019.014,E2 -24019.014} C_VEL
LIN {X 0,Y 147.571,Z 531.482,A -85,B 0,C 180,E1 -24021.784,E2 -24021.784} C_VEL
LIN {X 0,Y 148.003,Z 529.15,A -85,B 0,C 180,E1 -24025.705,E2 -24025.705} C_VEL
LIN {X 0,Y 148.691,Z 525.56,A -85,B 0,C 180,E1 -24029.999,E2 -24029.999} C_VEL
LIN {X 0,Y 149.915,Z 521.029,A -85,B 0,C 180,E1 -24034.031,E2 -24034.031} C_VEL
LIN {X 0,Y 151.981,Z 514.17,A -85,B 0,C 180,E1 -24038.642,E2 -24038.642} C_VEL
LIN {X 0,Y 154.434,Z 506.739,A -85,B 0,C 180,E1 -24042.482,E2 -24042.482} C_VEL
LIN {X 0,Y 156.895,Z 499.164,A -85,B 0,C 180,E1 -24045.589,E2 -24045.589} C_VEL
LIN {X 0,Y 159.81,Z 489.976,A -85,B 0,C 180,E1 -24048.591,E2 -24048.591} C_VEL
LIN {X 0,Y 162.777,Z 479.739,A -85,B 0,C 180,E1 -24051.197,E2 -24051.197} C_VEL
LIN {X 0,Y 165.767,Z 468.362,A -85,B 0,C 180,E1 -24053.418,E2 -24053.418} C_VEL
LIN {X 0,Y 168.094,Z 456.609,A -85,B 0,C 180,E1 -24055.208,E2 -24055.208} C_VEL
LIN {X 0,Y 169.83,Z 443.727,A -85,B 0,C 180,E1 -24056.661,E2 -24056.661} C_VEL
LIN {X 0,Y 171.45,Z 429.878,A -85,B 0,C 180,E1 -24057.615,E2 -24057.615} C_VEL
LIN {X 0,Y 174.608,Z 375.767,A -85,B 0,C 180,E1 -24059.649,E2 -24059.649} C_VEL
LIN {X 0,Y 169.053,Z 363.628,A -85,B 0,C 180,E1 -24061.639,E2 -24061.639} C_VEL
LIN {X 0,Y 162.065,Z 350.806,A -85,B 0,C 180,E1 -24064.282,E2 -24064.282} C_VEL
LIN {X 0,Y 155.555,Z 340.558,A -85,B 0,C 180,E1 -24066.954,E2 -24066.954} C_VEL
LIN {X 0,Y 153.244,Z 337.042,A -85,B 0,C 180,E1 -24067.978,E2 -24067.978} C_VEL
LIN {X 0,Y 150.788,Z 333.98,A -85,B 0,C 180,E1 -24069.078,E2 -24069.078} C_VEL
LIN {X 0,Y 150.135,Z 331.774,A -85,B 0,C 180,E1 -24069.498,E2 -24069.498} C_VEL
LIN {X 0,Y 150.121,Z 331.769,A -85,B 0,C 180,E1 -24075.394,E2 -24075.394} C_VEL
LIN {X 0,Y 150.135,Z 331.774,A -85,B 0,C 180,E1 -24079.054,E2 -24079.054} C_VEL
LIN {X 0,Y 150.171,Z 331.759,A -85,B 0,C 180,E1 -24082.708,E2 -24082.708} C_VEL
LIN {X 0,Y 150.209,Z 331.763,A -85,B 0,C 180,E1 -24087.368,E2 -24087.368} C_VEL
LIN {X 0,Y 150.236,Z 331.761,A -85,B 0,C 180,E1 -24092.72,E2 -24092.72} C_VEL
LIN {X 0,Y 150.344,Z 331.728,A -85,B 0,C 180,E1 -24099.209,E2 -24099.209} C_VEL
LIN {X 0,Y 150.356,Z 331.753,A -85,B 0,C 180,E1 -24103.713,E2 -24103.713} C_VEL
LIN {X 0,Y 150.604,Z 331.695,A -85,B 0,C 180,E1 -24109.242,E2 -24109.242} C_VEL
LIN {X 0,Y 150.679,Z 331.694,A -85,B 0,C 180,E1 -24111.957,E2 -24111.957} C_VEL
LIN {X 0,Y 151.21,Z 331.619,A -85,B 0,C 180,E1 -24120,E2 -24120} C_VEL
LIN {X 0,Y 150.737,Z 331.698,A -85,B 0,C 180,E1 -24128.041,E2 -24128.041} C_VEL
LIN {X 0,Y 150.601,Z 331.696,A -85,B 0,C 180,E1 -24131.491,E2 -24131.491} C_VEL
LIN {X 0,Y 150.357,Z 331.757,A -85,B 0,C 180,E1 -24136.288,E2 -24136.288} C_VEL
LIN {X 0,Y 150.347,Z 331.757,A -85,B 0,C 180,E1 -24140.793,E2 -24140.793} C_VEL
LIN {X 0,Y 150.241,Z 331.77,A -85,B 0,C 180,E1 -24147.283,E2 -24147.283} C_VEL
LIN {X 0,Y 150.214,Z 331.776,A -85,B 0,C 180,E1 -24152.635,E2 -24152.635} C_VEL
LIN {X 0,Y 150.208,Z 331.777,A -85,B 0,C 180,E1 -24157.464,E2 -24157.464} C_VEL
LIN {X 0,Y 150.179,Z 331.939,A -85,B 0,C 180,E1 -24160.051,E2 -24160.051} C_VEL
LIN {X 0,Y 151.172,Z 334.647,A -85,B 0,C 180,E1 -24160.607,E2 -24160.607} C_VEL
LIN {X 0,Y 153.321,Z 337.207,A -85,B 0,C 180,E1 -24161.557,E2 -24161.557} C_VEL
LIN {X 0,Y 155.576,Z 340.625,A -85,B 0,C 180,E1 -24162.557,E2 -24162.557} C_VEL
LIN {X 0,Y 161.221,Z 351.259,A -85,B 0,C 180,E1 -24164.993,E2 -24164.993} C_VEL
LIN {X 0,Y 166.11,Z 361.907,A -85,B 0,C 180,E1 -24166.984,E2 -24166.984} C_VEL
LIN {X 0,Y 170.454,Z 373.092,A -85,B 0,C 180,E1 -24168.709,E2 -24168.709} C_VEL
LIN {X 0,Y 172.276,Z 378.363,A -85,B 0,C 180,E1 -24169.425,E2 -24169.425} C_VEL
LIN {X 0,Y 173.575,Z 395.599,A -85,B 0,C 180,E1 -24170.593,E2 -24170.593} C_VEL
LIN {X 0,Y 171.114,Z 440.644,A -85,B 0,C 180,E1 -24172.344,E2 -24172.344} C_VEL
LIN {X 0,Y 169.596,Z 453.878,A -85,B 0,C 180,E1 -24173.255,E2 -24173.255} C_VEL
LIN {X 0,Y 167.437,Z 466.598,A -85,B 0,C 180,E1 -24174.568,E2 -24174.568} C_VEL
LIN {X 0,Y 164.773,Z 478.681,A -85,B 0,C 180,E1 -24176.327,E2 -24176.327} C_VEL
LIN {X 0,Y 161.729,Z 490.225,A -85,B 0,C 180,E1 -24178.571,E2 -24178.571} C_VEL
LIN {X 0,Y 158.754,Z 500.641,A -85,B 0,C 180,E1 -24181.223,E2 -24181.223} C_VEL
LIN {X 0,Y 155.999,Z 509.467,A -85,B 0,C 180,E1 -24184.086,E2 -24184.086} C_VEL
LIN {X 0,Y 154.123,Z 515.5,A -85,B 0,C 180,E1 -24186.486,E2 -24186.486} C_VEL
LIN {X 0,Y 151.613,Z 523.48,A -85,B 0,C 180,E1 -24190.364,E2 -24190.364} C_VEL
LIN {X 0,Y 149.894,Z 528.866,A -85,B 0,C 180,E1 -24193.663,E2 -24193.663} C_VEL
LIN {X 0,Y 148.906,Z 532.782,A -85,B 0,C 180,E1 -24196.589,E2 -24196.589} C_VEL
LIN {X 0,Y 147.742,Z 535.154,A -85,B 0,C 180,E1 -24198.637,E2 -24198.637} C_VEL
LIN {X 0,Y 144.402,Z 538.4,A -85,B 0,C 180,E1 -24202.07,E2 -24202.07} C_VEL
LIN {X 0,Y 141.817,Z 540.46,A -85,B 0,C 180,E1 -24204.986,E2 -24204.986} C_VEL
LIN {X 0,Y 140.747,Z 541.702,A -85,B 0,C 180,E1 -24207.311,E2 -24207.311} C_VEL
LIN {X 0,Y 140.665,Z 542.056,A -85,B 0,C 180,E1 -24208.106,E2 -24208.106} C_VEL
LIN {X 0,Y 140.747,Z 542.861,A -85,B 0,C 180,E1 -24210.002,E2 -24210.002} C_VEL
LIN {X 0,Y 140.59,Z 543.71,A -85,B 0,C 180,E1 -24212.867,E2 -24212.867} C_VEL
LIN {X 0,Y 140.622,Z 544.13,A -85,B 0,C 180,E1 -24215.738,E2 -24215.738} C_VEL
LIN {X 0,Y 141.424,Z 543.79,A -85,B 0,C 180,E1 -24221.467,E2 -24221.467} C_VEL
LIN {X 0,Y 142.246,Z 543.052,A -85,B 0,C 180,E1 -24224.304,E2 -24224.304} C_VEL
LIN {X 0,Y 143.354,Z 541.911,A -85,B 0,C 180,E1 -24227.108,E2 -24227.108} C_VEL
LIN {X 0,Y 146.817,Z 538.363,A -85,B 0,C 180,E1 -24232.518,E2 -24232.518} C_VEL
LIN {X 0,Y 150.199,Z 534.556,A -85,B 0,C 180,E1 -24236.394,E2 -24236.394} C_VEL
LIN {X 0,Y 154.133,Z 529.652,A -85,B 0,C 180,E1 -24240.105,E2 -24240.105} C_VEL
LIN {X 0,Y 158.728,Z 523.505,A -85,B 0,C 180,E1 -24243.606,E2 -24243.606} C_VEL
LIN {X 0,Y 164.096,Z 515.887,A -85,B 0,C 180,E1 -24246.842,E2 -24246.842} C_VEL
LIN {X 0,Y 169.913,Z 506.34,A -85,B 0,C 180,E1 -24249.876,E2 -24249.876} C_VEL
LIN {X 0,Y 175.181,Z 496.51,A -85,B 0,C 180,E1 -24252.221,E2 -24252.221} C_VEL
LIN {X 0,Y 180.191,Z 485.517,A -85,B 0,C 180,E1 -24254.202,E2 -24254.202} C_VEL
LIN {X 0,Y 184.236,Z 474.77,A -85,B 0,C 180,E1 -24255.664,E2 -24255.664} C_VEL
LIN {X 0,Y 188.145,Z 461.824,A -85,B 0,C 180,E1 -24256.949,E2 -24256.949} C_VEL
LIN {X 0,Y 190.908,Z 449.158,A -85,B 0,C 180,E1 -24257.831,E2 -24257.831} C_VEL
LIN {X 0,Y 192.744,Z 435.507,A -85,B 0,C 180,E1 -24258.442,E2 -24258.442} C_VEL
LIN {X 0,Y 194.686,Z 410.321,A -85,B 0,C 180,E1 -24259.233,E2 -24259.233} C_VEL
LIN {X 0,Y 190.706,Z 399.904,A -85,B 0,C 180,E1 -24261.564,E2 -24261.564} C_VEL
LIN {X 0,Y 186.325,Z 390.188,A -85,B 0,C 180,E1 -24264.305,E2 -24264.305} C_VEL
LIN {X 0,Y 181.478,Z 380.772,A -85,B 0,C 180,E1 -24267.7,E2 -24267.7} C_VEL
LIN {X 0,Y 178.284,Z 374.994,A -85,B 0,C 180,E1 -24270.239,E2 -24270.239} C_VEL
LIN {X 0,Y 176.664,Z 372.2,A -85,B 0,C 180,E1 -24271.647,E2 -24271.647} C_VEL
LIN {X 0,Y 173.854,Z 367.502,A -85,B 0,C 180,E1 -24274.352,E2 -24274.352} C_VEL
LIN {X 0,Y 170.189,Z 362.134,A -85,B 0,C 180,E1 -24278.547,E2 -24278.547} C_VEL
LIN {X 0,Y 167.659,Z 359.577,A -85,B 0,C 180,E1 -24282.15,E2 -24282.15} C_VEL
LIN {X 0,Y 166.425,Z 356.907,A -85,B 0,C 180,E1 -24284.696,E2 -24284.696} C_VEL
LIN {X 0,Y 163.974,Z 354.969,A -85,B 0,C 180,E1 -24292.612,E2 -24292.612} C_VEL
LIN {X 0,Y 164.132,Z 354.752,A -85,B 0,C 180,E1 -24298.773,E2 -24298.773} C_VEL
LIN {X 0,Y 166.757,Z 356.996,A -85,B 0,C 180,E1 -24306.465,E2 -24306.465} C_VEL
LIN {X 0,Y 168.605,Z 360.543,A -85,B 0,C 180,E1 -24309.867,E2 -24309.867} C_VEL
LIN {X 0,Y 170.583,Z 362.53,A -85,B 0,C 180,E1 -24312.491,E2 -24312.491} C_VEL
LIN {X 0,Y 173.15,Z 366.247,A -85,B 0,C 180,E1 -24315.448,E2 -24315.448} C_VEL
LIN {X 0,Y 174.217,Z 367.566,A -85,B 0,C 180,E1 -24316.515,E2 -24316.515} C_VEL
LIN {X 0,Y 176.898,Z 371.245,A -85,B 0,C 180,E1 -24318.982,E2 -24318.982} C_VEL
LIN {X 0,Y 180.794,Z 377.041,A -85,B 0,C 180,E1 -24322.122,E2 -24322.122} C_VEL
LIN {X 0,Y 185.022,Z 383.525,A -85,B 0,C 180,E1 -24325.072,E2 -24325.072} C_VEL
LIN {X 0,Y 189.692,Z 391.457,A -85,B 0,C 180,E1 -24327.963,E2 -24327.963} C_VEL
LIN {X 0,Y 194.686,Z 400.759,A -85,B 0,C 180,E1 -24330.732,E2 -24330.732} C_VEL
LIN {X 0,Y 195.175,Z 401.86,A -85,B 0,C 180,E1 -24330.997,E2 -24330.997} C_VEL
LIN {X 0,Y 192.752,Z 431.814,A -85,B 0,C 180,E1 -24331.987,E2 -24331.987} C_VEL
LIN {X 0,Y 190.635,Z 445.214,A -85,B 0,C 180,E1 -24332.752,E2 -24332.752} C_VEL
LIN {X 0,Y 187.932,Z 456.644,A -85,B 0,C 180,E1 -24333.687,E2 -24333.687} C_VEL
LIN {X 0,Y 184.456,Z 468.463,A -85,B 0,C 180,E1 -24335.094,E2 -24335.094} C_VEL
LIN {X 0,Y 180.622,Z 478.593,A -85,B 0,C 180,E1 -24336.628,E2 -24336.628} C_VEL
LIN {X 0,Y 175.83,Z 489.384,A -85,B 0,C 180,E1 -24338.791,E2 -24338.791} C_VEL
LIN {X 0,Y 170.949,Z 498.538,A -85,B 0,C 180,E1 -24341.131,E2 -24341.131} C_VEL
LIN {X 0,Y 165.803,Z 506.891,A -85,B 0,C 180,E1 -24343.896,E2 -24343.896} C_VEL
LIN {X 0,Y 160.478,Z 514.527,A -85,B 0,C 180,E1 -24347.248,E2 -24347.248} C_VEL
LIN {X 0,Y 155.742,Z 520.624,A -85,B 0,C 180,E1 -24350.819,E2 -24350.819} C_VEL
LIN {X 0,Y 151.595,Z 525.411,A -85,B 0,C 180,E1 -24354.583,E2 -24354.583} C_VEL
LIN {X 0,Y 147.896,Z 529.25,A -85,B 0,C 180,E1 -24358.799,E2 -24358.799} C_VEL
LIN {X 0,Y 146.154,Z 530.887,A -85,B 0,C 180,E1 -24361.257,E2 -24361.257} C_VEL
LIN {X 0,Y 144.46,Z 532.252,A -85,B 0,C 180,E1 -24364.032,E2 -24364.032} C_VEL
LIN {X 0,Y 143.135,Z 533.207,A -85,B 0,C 180,E1 -24366.87,E2 -24366.87} C_VEL
LIN {X 0,Y 141.939,Z 533.82,A -85,B 0,C 180,E1 -24370.181,E2 -24370.181} C_VEL
LIN {X 0,Y 140.751,Z 533.614,A -85,B 0,C 180,E1 -24375.541,E2 -24375.541} C_VEL
LIN {X 0,Y 140.478,Z 532.938,A -85,B 0,C 180,E1 -24378.455,E2 -24378.455} C_VEL
LIN {X 0,Y 140.454,Z 531.872,A -85,B 0,C 180,E1 -24381.365,E2 -24381.365} C_VEL
LIN {X 0,Y 140.926,Z 529.353,A -85,B 0,C 180,E1 -24385.865,E2 -24385.865} C_VEL
LIN {X 0,Y 141.596,Z 526.065,A -85,B 0,C 180,E1 -24389.998,E2 -24389.998} C_VEL
LIN {X 0,Y 142.821,Z 521.61,A -85,B 0,C 180,E1 -24394.231,E2 -24394.231} C_VEL
LIN {X 0,Y 144.989,Z 514.866,A -85,B 0,C 180,E1 -24399.062,E2 -24399.062} C_VEL
LIN {X 0,Y 147.536,Z 507.526,A -85,B 0,C 180,E1 -24403.076,E2 -24403.076} C_VEL
LIN {X 0,Y 150.665,Z 498.419,A -85,B 0,C 180,E1 -24406.949,E2 -24406.949} C_VEL
LIN {X 0,Y 154.105,Z 487.876,A -85,B 0,C 180,E1 -24410.347,E2 -24410.347} C_VEL
LIN {X 0,Y 157.279,Z 477.14,A -85,B 0,C 180,E1 -24413.014,E2 -24413.014} C_VEL
LIN {X 0,Y 160.112,Z 466.662,A -85,B 0,C 180,E1 -24414.99,E2 -24414.99} C_VEL
LIN {X 0,Y 162.478,Z 454.181,A -85,B 0,C 180,E1 -24416.837,E2 -24416.837} C_VEL
LIN {X 0,Y 164.318,Z 440.707,A -85,B 0,C 180,E1 -24418.275,E2 -24418.275} C_VEL
LIN {X 0,Y 165.764,Z 427.899,A -85,B 0,C 180,E1 -24419.06,E2 -24419.06} C_VEL
LIN {X 0,Y 168.682,Z 377.66,A -85,B 0,C 180,E1 -24420.997,E2 -24420.997} C_VEL
LIN {X 0,Y 162.964,Z 365.274,A -85,B 0,C 180,E1 -24423.205,E2 -24423.205} C_VEL
LIN {X 0,Y 156.901,Z 354.261,A -85,B 0,C 180,E1 -24425.674,E2 -24425.674} C_VEL
LIN {X 0,Y 151.507,Z 345.666,A -85,B 0,C 180,E1 -24428.049,E2 -24428.049} C_VEL
LIN {X 0,Y 148.41,Z 341.27,A -85,B 0,C 180,E1 -24429.501,E2 -24429.501} C_VEL
LIN {X 0,Y 146.296,Z 337.869,A -85,B 0,C 180,E1 -24430.577,E2 -24430.577} C_VEL
LIN {X 0,Y 143.91,Z 335.221,A -85,B 0,C 180,E1 -24431.771,E2 -24431.771} C_VEL
LIN {X 0,Y 143.043,Z 332.657,A -85,B 0,C 180,E1 -24432.364,E2 -24432.364} C_VEL
LIN {X 0,Y 143.052,Z 332.664,A -85,B 0,C 180,E1 -24437.468,E2 -24437.468} C_VEL
LIN {X 0,Y 143.067,Z 332.638,A -85,B 0,C 180,E1 -24441.808,E2 -24441.808} C_VEL
LIN {X 0,Y 143.176,Z 332.638,A -85,B 0,C 180,E1 -24447.32,E2 -24447.32} C_VEL
LIN {X 0,Y 143.183,Z 332.632,A -85,B 0,C 180,E1 -24452.064,E2 -24452.064} C_VEL
LIN {X 0,Y 143.27,Z 332.61,A -85,B 0,C 180,E1 -24458.748,E2 -24458.748} C_VEL
LIN {X 0,Y 143.29,Z 332.627,A -85,B 0,C 180,E1 -24462.886,E2 -24462.886} C_VEL
LIN {X 0,Y 143.531,Z 332.578,A -85,B 0,C 180,E1 -24468.705,E2 -24468.705} C_VEL
LIN {X 0,Y 143.605,Z 332.57,A -85,B 0,C 180,E1 -24471.558,E2 -24471.558} C_VEL
LIN {X 0,Y 144.169,Z 332.495,A -85,B 0,C 180,E1 -24480,E2 -24480} C_VEL
LIN {X 0,Y 143.656,Z 332.576,A -85,B 0,C 180,E1 -24488.44,E2 -24488.44} C_VEL
LIN {X 0,Y 143.543,Z 332.575,A -85,B 0,C 180,E1 -24491.713,E2 -24491.713} C_VEL
LIN {X 0,Y 143.297,Z 332.631,A -85,B 0,C 180,E1 -24497.114,E2 -24497.114} C_VEL
LIN {X 0,Y 143.273,Z 332.636,A -85,B 0,C 180,E1 -24501.256,E2 -24501.256} C_VEL
LIN {X 0,Y 143.187,Z 332.652,A -85,B 0,C 180,E1 -24507.939,E2 -24507.939} C_VEL
LIN {X 0,Y 143.164,Z 332.652,A -85,B 0,C 180,E1 -24513.436,E2 -24513.436} C_VEL
LIN {X 0,Y 143.161,Z 332.662,A -85,B 0,C 180,E1 -24517.213,E2 -24517.213} C_VEL
LIN {X 0,Y 144.191,Z 335.574,A -85,B 0,C 180,E1 -24517.874,E2 -24517.874} C_VEL
LIN {X 0,Y 146.368,Z 337.988,A -85,B 0,C 180,E1 -24518.956,E2 -24518.956} C_VEL
LIN {X 0,Y 148.507,Z 341.375,A -85,B 0,C 180,E1 -24520.04,E2 -24520.04} C_VEL
LIN {X 0,Y 152.097,Z 346.818,A -85,B 0,C 180,E1 -24521.735,E2 -24521.735} C_VEL
LIN {X 0,Y 157.866,Z 358.036,A -85,B 0,C 180,E1 -24524.357,E2 -24524.357} C_VEL
LIN {X 0,Y 162.894,Z 370.033,A -85,B 0,C 180,E1 -24526.54,E2 -24526.54} C_VEL
LIN {X 0,Y 166.661,Z 380.779,A -85,B 0,C 180,E1 -24528.145,E2 -24528.145} C_VEL
LIN {X 0,Y 167.729,Z 397.333,A -85,B 0,C 180,E1 -24529.289,E2 -24529.289} C_VEL
LIN {X 0,Y 165.164,Z 440.946,A -85,B 0,C 180,E1 -24531.028,E2 -24531.028} C_VEL
LIN {X 0,Y 163.47,Z 454.761,A -85,B 0,C 180,E1 -24532.026,E2 -24532.026} C_VEL
LIN {X 0,Y 161.236,Z 467.135,A -85,B 0,C 180,E1 -24533.375,E2 -24533.375} C_VEL
LIN {X 0,Y 158.468,Z 479.015,A -85,B 0,C 180,E1 -24535.182,E2 -24535.182} C_VEL
LIN {X 0,Y 155.305,Z 490.451,A -85,B 0,C 180,E1 -24537.497,E2 -24537.497} C_VEL
LIN {X 0,Y 152.193,Z 500.762,A -85,B 0,C 180,E1 -24540.239,E2 -24540.239} C_VEL
LIN {X 0,Y 149.006,Z 510.341,A -85,B 0,C 180,E1 -24543.533,E2 -24543.533} C_VEL
LIN {X 0,Y 147.127,Z 516.271,A -85,B 0,C 180,E1 -24546.046,E2 -24546.046} C_VEL
LIN {X 0,Y 144.508,Z 523.998,A -85,B 0,C 180,E1 -24550.098,E2 -24550.098} C_VEL
LIN {X 0,Y 142.483,Z 530.192,A -85,B 0,C 180,E1 -24554.261,E2 -24554.261} C_VEL
LIN {X 0,Y 141.33,Z 535.109,A -85,B 0,C 180,E1 -24558.528,E2 -24558.528} C_VEL
LIN {X 0,Y 140.761,Z 538.874,A -85,B 0,C 180,E1 -24562.831,E2 -24562.831} C_VEL
LIN {X 0,Y 140.665,Z 542.056,A -85,B 0,C 180,E1 -24568.106,E2 -24568.106} C_VEL
LIN {X 0,Y 139.975,Z 543.001,A -85,B 0,C 180,E1 -24570.468,E2 -24570.468} C_VEL
LIN {X 0,Y 138.363,Z 543.581,A -85,B 0,C 180,E1 -24572.812,E2 -24572.812} C_VEL
LIN {X 0,Y 134.821,Z 543.963,A -85,B 0,C 180,E1 -24577.633,E2 -24577.633} C_VEL
LIN {X 0,Y 134.12,Z 543.825,A -85,B 0,C 180,E1 -24580.167,E2 -24580.167} C_VEL
LIN {X 0,Y 134.206,Z 543.68,A -85,B 0,C 180,E1 -24581.019,E2 -24581.019} C_VEL
LIN {X 0,Y 135.352,Z 542.849,A -85,B 0,C 180,E1 -24585.049,E2 -24585.049} C_VEL
LIN {X 0,Y 136.552,Z 541.75,A -85,B 0,C 180,E1 -24587.989,E2 -24587.989} C_VEL
LIN {X 0,Y 138.236,Z 540.214,A -85,B 0,C 180,E1 -24590.849,E2 -24590.849} C_VEL
LIN {X 0,Y 141.339,Z 537.145,A -85,B 0,C 180,E1 -24595.004,E2 -24595.004} C_VEL
LIN {X 0,Y 145.985,Z 532.049,A -85,B 0,C 180,E1 -24599.751,E2 -24599.751} C_VEL
LIN {X 0,Y 151.152,Z 525.787,A -85,B 0,C 180,E1 -24603.916,E2 -24603.916} C_VEL
LIN {X 0,Y 156.541,Z 518.762,A -85,B 0,C 180,E1 -24607.309,E2 -24607.309} C_VEL
LIN {X 0,Y 162.444,Z 510.006,A -85,B 0,C 180,E1 -24610.464,E2 -24610.464} C_VEL
LIN {X 0,Y 168.325,Z 500.086,A -85,B 0,C 180,E1 -24613.134,E2 -24613.134} C_VEL
LIN {X 0,Y 172.898,Z 491.235,A -85,B 0,C 180,E1 -24614.933,E2 -24614.933} C_VEL
LIN {X 0,Y 176.914,Z 481.91,A -85,B 0,C 180,E1 -24616.469,E2 -24616.469} C_VEL
LIN {X 0,Y 181.232,Z 470.262,A -85,B 0,C 180,E1 -24617.873,E2 -24617.873} C_VEL
LIN {X 0,Y 184.966,Z 456.903,A -85,B 0,C 180,E1 -24619.041,E2 -24619.041} C_VEL
LIN {X 0,Y 187.514,Z 443.733,A -85,B 0,C 180,E1 -24619.832,E2 -24619.832} C_VEL
LIN {X 0,Y 189.122,Z 428.566,A -85,B 0,C 180,E1 -24620.379,E2 -24620.379} C_VEL
LIN {X 0,Y 190.338,Z 412.761,A -85,B 0,C 180,E1 -24620.882,E2 -24620.882} C_VEL
LIN {X 0,Y 186.952,Z 403.822,A -85,B 0,C 180,E1 -24623.024,E2 -24623.024} C_VEL
LIN {X 0,Y 182.97,Z 394.68,A -85,B 0,C 180,E1 -24625.729,E2 -24625.729} C_VEL
LIN {X 0,Y 178.66,Z 385.961,A -85,B 0,C 180,E1 -24628.997,E2 -24628.997} C_VEL
LIN {X 0,Y 175.052,Z 379.052,A -85,B 0,C 180,E1 -24632.159,E2 -24632.159} C_VEL
LIN {X 0,Y 171.74,Z 373.453,A -85,B 0,C 180,E1 -24635.522,E2 -24635.522} C_VEL
LIN {X 0,Y 168.637,Z 368.819,A -85,B 0,C 180,E1 -24639.333,E2 -24639.333} C_VEL
LIN {X 0,Y 166.315,Z 366.185,A -85,B 0,C 180,E1 -24642.913,E2 -24642.913} C_VEL
LIN {X 0,Y 165.276,Z 363.849,A -85,B 0,C 180,E1 -24645.218,E2 -24645.218} C_VEL
LIN {X 0,Y 163.106,Z 362.033,A -85,B 0,C 180,E1 -24652.573,E2 -24652.573} C_VEL
LIN {X 0,Y 163.26,Z 361.79,A -85,B 0,C 180,E1 -24658.766,E2 -24658.766} C_VEL
LIN {X 0,Y 165.64,Z 364.002,A -85,B 0,C 180,E1 -24666.051,E2 -24666.051} C_VEL
LIN {X 0,Y 167.447,Z 367.512,A -85,B 0,C 180,E1 -24669.512,E2 -24669.512} C_VEL
LIN {X 0,Y 169.116,Z 369.281,A -85,B 0,C 180,E1 -24671.84,E2 -24671.84} C_VEL
LIN {X 0,Y 171.8,Z 373.139,A -85,B 0,C 180,E1 -24675.05,E2 -24675.05} C_VEL
LIN {X 0,Y 175.617,Z 378.739,A -85,B 0,C 180,E1 -24678.785,E2 -24678.785} C_VEL
LIN {X 0,Y 178.451,Z 382.994,A -85,B 0,C 180,E1 -24681.156,E2 -24681.156} C_VEL
LIN {X 0,Y 182.496,Z 389.493,A -85,B 0,C 180,E1 -24684.153,E2 -24684.153} C_VEL
LIN {X 0,Y 186.712,Z 396.93,A -85,B 0,C 180,E1 -24686.927,E2 -24686.927} C_VEL
LIN {X 0,Y 190.786,Z 404.8,A -85,B 0,C 180,E1 -24689.347,E2 -24689.347} C_VEL
LIN {X 0,Y 188.519,Z 432.126,A -85,B 0,C 180,E1 -24690.276,E2 -24690.276} C_VEL
LIN {X 0,Y 186.281,Z 445.768,A -85,B 0,C 180,E1 -24691.059,E2 -24691.059} C_VEL
LIN {X 0,Y 183.373,Z 457.574,A -85,B 0,C 180,E1 -24692.038,E2 -24692.038} C_VEL
LIN {X 0,Y 179.548,Z 469.786,A -85,B 0,C 180,E1 -24693.526,E2 -24693.526} C_VEL
LIN {X 0,Y 175.231,Z 480.485,A -85,B 0,C 180,E1 -24695.195,E2 -24695.195} C_VEL
LIN {X 0,Y 170.275,Z 490.989,A -85,B 0,C 180,E1 -24697.388,E2 -24697.388} C_VEL
LIN {X 0,Y 164.91,Z 500.336,A -85,B 0,C 180,E1 -24699.904,E2 -24699.904} C_VEL
LIN {X 0,Y 158.897,Z 509.378,A -85,B 0,C 180,E1 -24703.13,E2 -24703.13} C_VEL
LIN {X 0,Y 153.469,Z 516.601,A -85,B 0,C 180,E1 -24706.613,E2 -24706.613} C_VEL
LIN {X 0,Y 148.603,Z 522.305,A -85,B 0,C 180,E1 -24710.321,E2 -24710.321} C_VEL
LIN {X 0,Y 144.371,Z 526.76,A -85,B 0,C 180,E1 -24714.255,E2 -24714.255} C_VEL
LIN {X 0,Y 141.409,Z 529.604,A -85,B 0,C 180,E1 -24717.66,E2 -24717.66} C_VEL
LIN {X 0,Y 137.939,Z 532.411,A -85,B 0,C 180,E1 -24722.705,E2 -24722.705} C_VEL
LIN {X 0,Y 136.466,Z 533.398,A -85,B 0,C 180,E1 -24725.668,E2 -24725.668} C_VEL
LIN {X 0,Y 134.964,Z 534.096,A -85,B 0,C 180,E1 -24729.605,E2 -24729.605} C_VEL
LIN {X 0,Y 133.749,Z 533.931,A -85,B 0,C 180,E1 -24734.766,E2 -24734.766} C_VEL
LIN {X 0,Y 133.425,Z 533.285,A -85,B 0,C 180,E1 -24737.835,E2 -24737.835} C_VEL
LIN {X 0,Y 133.337,Z 532.251,A -85,B 0,C 180,E1 -24740.9,E2 -24740.9} C_VEL
LIN {X 0,Y 133.857,Z 529.576,A -85,B 0,C 180,E1 -24746.005,E2 -24746.005} C_VEL
LIN {X 0,Y 134.499,Z 526.57,A -85,B 0,C 180,E1 -24749.998,E2 -24749.998} C_VEL
LIN {X 0,Y 135.733,Z 522.188,A -85,B 0,C 180,E1 -24754.453,E2 -24754.453} C_VEL
LIN {X 0,Y 137.641,Z 516.615,A -85,B 0,C 180,E1 -24758.81,E2 -24758.81} C_VEL
LIN {X 0,Y 140.157,Z 509.663,A -85,B 0,C 180,E1 -24763.039,E2 -24763.039} C_VEL
LIN {X 0,Y 143.307,Z 500.953,A -85,B 0,C 180,E1 -24767.111,E2 -24767.111} C_VEL
LIN {X 0,Y 146.488,Z 492.023,A -85,B 0,C 180,E1 -24770.353,E2 -24770.353} C_VEL
LIN {X 0,Y 149.678,Z 482.209,A -85,B 0,C 180,E1 -24773.154,E2 -24773.154} C_VEL
LIN {X 0,Y 152.875,Z 471.344,A -85,B 0,C 180,E1 -24775.528,E2 -24775.528} C_VEL
LIN {X 0,Y 155.318,Z 461.177,A -85,B 0,C 180,E1 -24777.266,E2 -24777.266} C_VEL
LIN {X 0,Y 157.373,Z 449.165,A -85,B 0,C 180,E1 -24778.871,E2 -24778.871} C_VEL
LIN {X 0,Y 158.869,Z 438.136,A -85,B 0,C 180,E1 -24779.908,E2 -24779.908} C_VEL
LIN {X 0,Y 160.255,Z 424.69,A -85,B 0,C 180,E1 -24780.655,E2 -24780.655} C_VEL
LIN {X 0,Y 162.905,Z 379.563,A -85,B 0,C 180,E1 -24782.427,E2 -24782.427} C_VEL
LIN {X 0,Y 157.374,Z 367.831,A -85,B 0,C 180,E1 -24784.717,E2 -24784.717} C_VEL
LIN {X 0,Y 151.416,Z 356.925,A -85,B 0,C 180,E1 -24787.358,E2 -24787.358} C_VEL
LIN {X 0,Y 145.196,Z 347.227,A -85,B 0,C 180,E1 -24790.372,E2 -24790.372} C_VEL
LIN {X 0,Y 141.869,Z 342.595,A -85,B 0,C 180,E1 -24792.127,E2 -24792.127} C_VEL
LIN {X 0,Y 139.626,Z 339.289,A -85,B 0,C 180,E1 -24793.404,E2 -24793.404} C_VEL
LIN {X 0,Y 138.986,Z 338.5,A -85,B 0,C 180,E1 -24793.77,E2 -24793.77} C_VEL
LIN {X 0,Y 136.907,Z 336.305,A -85,B 0,C 180,E1 -24794.972,E2 -24794.972} C_VEL
LIN {X 0,Y 136.038,Z 334.016,A -85,B 0,C 180,E1 -24795.609,E2 -24795.609} C_VEL
LIN {X 0,Y 135.983,Z 333.531,A -85,B 0,C 180,E1 -24795.768,E2 -24795.768} C_VEL
LIN {X 0,Y 136.016,Z 333.516,A -85,B 0,C 180,E1 -24801.681,E2 -24801.681} C_VEL
LIN {X 0,Y 136.05,Z 333.536,A -85,B 0,C 180,E1 -24805.739,E2 -24805.739} C_VEL
LIN {X 0,Y 136.139,Z 333.511,A -85,B 0,C 180,E1 -24812.315,E2 -24812.315} C_VEL
LIN {X 0,Y 136.236,Z 333.484,A -85,B 0,C 180,E1 -24818.832,E2 -24818.832} C_VEL
LIN {X 0,Y 136.261,Z 333.512,A -85,B 0,C 180,E1 -24825.056,E2 -24825.056} C_VEL
LIN {X 0,Y 136.426,Z 333.466,A -85,B 0,C 180,E1 -24828.166,E2 -24828.166} C_VEL
LIN {X 0,Y 136.534,Z 333.446,A -85,B 0,C 180,E1 -24831.117,E2 -24831.117} C_VEL
LIN {X 0,Y 137.126,Z 333.371,A -85,B 0,C 180,E1 -24840,E2 -24840} C_VEL
LIN {X 0,Y 136.584,Z 333.45,A -85,B 0,C 180,E1 -24848.88,E2 -24848.88} C_VEL
LIN {X 0,Y 136.487,Z 333.454,A -85,B 0,C 180,E1 -24851.955,E2 -24851.955} C_VEL
LIN {X 0,Y 136.237,Z 333.509,A -85,B 0,C 180,E1 -24858.031,E2 -24858.031} C_VEL
LIN {X 0,Y 136.194,Z 333.516,A -85,B 0,C 180,E1 -24861.75,E2 -24861.75} C_VEL
LIN {X 0,Y 136.112,Z 333.533,A -85,B 0,C 180,E1 -24868.63,E2 -24868.63} C_VEL
LIN {X 0,Y 136.091,Z 333.533,A -85,B 0,C 180,E1 -24873.869,E2 -24873.869} C_VEL
LIN {X 0,Y 136.976,Z 336.245,A -85,B 0,C 180,E1 -24874.56,E2 -24874.56} C_VEL
LIN {X 0,Y 139.049,Z 338.492,A -85,B 0,C 180,E1 -24875.762,E2 -24875.762} C_VEL
LIN {X 0,Y 139.814,Z 339.501,A -85,B 0,C 180,E1 -24876.203,E2 -24876.203} C_VEL
LIN {X 0,Y 141.992,Z 342.693,A -85,B 0,C 180,E1 -24877.436,E2 -24877.436} C_VEL
LIN {X 0,Y 147.546,Z 350.762,A -85,B 0,C 180,E1 -24880.302,E2 -24880.302} C_VEL
LIN {X 0,Y 153.549,Z 362.975,A -85,B 0,C 180,E1 -24883.255,E2 -24883.255} C_VEL
LIN {X 0,Y 158.24,Z 374.519,A -85,B 0,C 180,E1 -24885.439,E2 -24885.439} C_VEL
LIN {X 0,Y 161.063,Z 382.742,A -85,B 0,C 180,E1 -24886.733,E2 -24886.733} C_VEL
LIN {X 0,Y 161.998,Z 398.069,A -85,B 0,C 180,E1 -24887.843,E2 -24887.843} C_VEL
LIN {X 0,Y 159.384,Z 440.529,A -85,B 0,C 180,E1 -24889.573,E2 -24889.573} C_VEL
LIN {X 0,Y 157.653,Z 454.211,A -85,B 0,C 180,E1 -24890.577,E2 -24890.577} C_VEL
LIN {X 0,Y 155.306,Z 466.603,A -85,B 0,C 180,E1 -24891.937,E2 -24891.937} C_VEL
LIN {X 0,Y 152.617,Z 477.744,A -85,B 0,C 180,E1 -24893.64,E2 -24893.64} C_VEL
LIN {X 0,Y 149.701,Z 488.062,A -85,B 0,C 180,E1 -24895.714,E2 -24895.714} C_VEL
LIN {X 0,Y 146.332,Z 498.758,A -85,B 0,C 180,E1 -24898.515,E2 -24898.515} C_VEL
LIN {X 0,Y 143.389,Z 507.497,A -85,B 0,C 180,E1 -24901.456,E2 -24901.456} C_VEL
LIN {X 0,Y 140.538,Z 515.632,A -85,B 0,C 180,E1 -24904.898,E2 -24904.898} C_VEL
LIN {X 0,Y 137.819,Z 523.382,A -85,B 0,C 180,E1 -24909.088,E2 -24909.088} C_VEL
LIN {X 0,Y 135.616,Z 529.641,A -85,B 0,C 180,E1 -24913.442,E2 -24913.442} C_VEL
LIN {X 0,Y 134.331,Z 534.618,A -85,B 0,C 180,E1 -24917.922,E2 -24917.922} C_VEL
LIN {X 0,Y 133.691,Z 538.441,A -85,B 0,C 180,E1 -24922.45,E2 -24922.45} C_VEL
LIN {X 0,Y 133.569,Z 541.775,A -85,B 0,C 180,E1 -24928.158,E2 -24928.158} C_VEL
LIN {X 0,Y 133.571,Z 542.962,A -85,B 0,C 180,E1 -24931.358,E2 -24931.358} C_VEL
LIN {X 0,Y 133.549,Z 543.852,A -85,B 0,C 180,E1 -24936.043,E2 -24936.043} C_VEL
LIN {X 0,Y 134.206,Z 543.68,A -85,B 0,C 180,E1 -24941.019,E2 -24941.019} C_VEL
LIN {X 0,Y 134.191,Z 543.277,A -85,B 0,C 180,E1 -24943.53,E2 -24943.53} C_VEL
LIN {X 0,Y 132.889,Z 541.957,A -85,B 0,C 180,E1 -24947.707,E2 -24947.707} C_VEL
LIN {X 0,Y 132.272,Z 540.065,A -85,B 0,C 180,E1 -24951.901,E2 -24951.901} C_VEL
LIN {X 0,Y 133.312,Z 538.524,A -85,B 0,C 180,E1 -24954.328,E2 -24954.328} C_VEL
LIN {X 0,Y 137.588,Z 534.474,A -85,B 0,C 180,E1 -24959.031,E2 -24959.031} C_VEL
LIN {X 0,Y 142.018,Z 529.693,A -85,B 0,C 180,E1 -24962.982,E2 -24962.982} C_VEL
LIN {X 0,Y 147.12,Z 523.682,A -85,B 0,C 180,E1 -24966.666,E2 -24966.666} C_VEL
LIN {X 0,Y 152.983,Z 516.222,A -85,B 0,C 180,E1 -24970.029,E2 -24970.029} C_VEL
LIN {X 0,Y 158.192,Z 508.637,A -85,B 0,C 180,E1 -24972.65,E2 -24972.65} C_VEL
LIN {X 0,Y 163.807,Z 499.463,A -85,B 0,C 180,E1 -24975.067,E2 -24975.067} C_VEL
LIN {X 0,Y 168.535,Z 490.545,A -85,B 0,C 180,E1 -24976.867,E2 -24976.867} C_VEL
LIN {X 0,Y 172.763,Z 481.128,A -85,B 0,C 180,E1 -24978.375,E2 -24978.375} C_VEL
LIN {X 0,Y 177.218,Z 469.283,A -85,B 0,C 180,E1 -24979.766,E2 -24979.766} C_VEL
LIN {X 0,Y 180.744,Z 457.001,A -85,B 0,C 180,E1 -24980.828,E2 -24980.828} C_VEL
LIN {X 0,Y 183.39,Z 443.978,A -85,B 0,C 180,E1 -24981.612,E2 -24981.612} C_VEL
LIN {X 0,Y 185.024,Z 429.615,A -85,B 0,C 180,E1 -24982.138,E2 -24982.138} C_VEL
LIN {X 0,Y 186.153,Z 415.355,A -85,B 0,C 180,E1 -24982.597,E2 -24982.597} C_VEL
LIN {X 0,Y 183.227,Z 407.362,A -85,B 0,C 180,E1 -24984.623,E2 -24984.623} C_VEL
LIN {X 0,Y 179.051,Z 397.613,A -85,B 0,C 180,E1 -24987.745,E2 -24987.745} C_VEL
LIN {X 0,Y 175.077,Z 389.282,A -85,B 0,C 180,E1 -24991.121,E2 -24991.121} C_VEL
LIN {X 0,Y 172.497,Z 384.42,A -85,B 0,C 180,E1 -24993.608,E2 -24993.608} C_VEL
LIN {X 0,Y 169.923,Z 379.728,A -85,B 0,C 180,E1 -24996.46,E2 -24996.46} C_VEL
LIN {X 0,Y 167.309,Z 375.618,A -85,B 0,C 180,E1 -24999.884,E2 -24999.884} C_VEL
LIN {X 0,Y 165.068,Z 372.934,A -85,B 0,C 180,E1 -25003.545,E2 -25003.545} C_VEL
LIN {X 0,Y 164.14,Z 370.788,A -85,B 0,C 180,E1 -25005.747,E2 -25005.747} C_VEL
LIN {X 0,Y 162.118,Z 368.968,A -85,B 0,C 180,E1 -25013.778,E2 -25013.778} C_VEL
LIN {X 0,Y 162.386,Z 368.843,A -85,B 0,C 180,E1 -25018.76,E2 -25018.76} C_VEL
LIN {X 0,Y 164.48,Z 370.94,A -85,B 0,C 180,E1 -25025.517,E2 -25025.517} C_VEL
LIN {X 0,Y 166.276,Z 374.438,A -85,B 0,C 180,E1 -25029.12,E2 -25029.12} C_VEL
LIN {X 0,Y 167.679,Z 376.014,A -85,B 0,C 180,E1 -25031.177,E2 -25031.177} C_VEL
LIN {X 0,Y 170.797,Z 380.741,A -85,B 0,C 180,E1 -25035.047,E2 -25035.047} C_VEL
LIN {X 0,Y 173.901,Z 385.481,A -85,B 0,C 180,E1 -25038.176,E2 -25038.176} C_VEL
LIN {X 0,Y 176.998,Z 390.328,A -85,B 0,C 180,E1 -25040.862,E2 -25040.862} C_VEL
LIN {X 0,Y 181.616,Z 398.231,A -85,B 0,C 180,E1 -25044.353,E2 -25044.353} C_VEL
LIN {X 0,Y 186.345,Z 407.405,A -85,B 0,C 180,E1 -25047.492,E2 -25047.492} C_VEL
LIN {X 0,Y 186.679,Z 408.027,A -85,B 0,C 180,E1 -25047.695,E2 -25047.695} C_VEL
LIN {X 0,Y 184.434,Z 432.656,A -85,B 0,C 180,E1 -25048.5,E2 -25048.5} C_VEL
LIN {X 0,Y 182.088,Z 446.41,A -85,B 0,C 180,E1 -25049.296,E2 -25049.296} C_VEL
LIN {X 0,Y 179.034,Z 458.209,A -85,B 0,C 180,E1 -25050.275,E2 -25050.275} C_VEL
LIN {X 0,Y 175.354,Z 469.563,A -85,B 0,C 180,E1 -25051.651,E2 -25051.651} C_VEL
LIN {X 0,Y 171.154,Z 479.746,A -85,B 0,C 180,E1 -25053.211,E2 -25053.211} C_VEL
LIN {X 0,Y 165.951,Z 490.428,A -85,B 0,C 180,E1 -25055.389,E2 -25055.389} C_VEL
LIN {X 0,Y 160.343,Z 499.969,A -85,B 0,C 180,E1 -25057.911,E2 -25057.911} C_VEL
LIN {X 0,Y 154.011,Z 509.118,A -85,B 0,C 180,E1 -25061.153,E2 -25061.153} C_VEL
LIN {X 0,Y 148.255,Z 516.452,A -85,B 0,C 180,E1 -25064.677,E2 -25064.677} C_VEL
LIN {X 0,Y 143.074,Z 522.26,A -85,B 0,C 180,E1 -25068.459,E2 -25068.459} C_VEL
LIN {X 0,Y 138.502,Z 526.788,A -85,B 0,C 180,E1 -25072.488,E2 -25072.488} C_VEL
LIN {X 0,Y 134.939,Z 529.981,A -85,B 0,C 180,E1 -25076.441,E2 -25076.441} C_VEL
LIN {X 0,Y 131.497,Z 532.57,A -85,B 0,C 180,E1 -25081.247,E2 -25081.247} C_VEL
LIN {X 0,Y 129.855,Z 533.589,A -85,B 0,C 180,E1 -25084.342,E2 -25084.342} C_VEL
LIN {X 0,Y 127.524,Z 534.441,A -85,B 0,C 180,E1 -25090.689,E2 -25090.689} C_VEL
LIN {X 0,Y 126.783,Z 534.248,A -85,B 0,C 180,E1 -25093.907,E2 -25093.907} C_VEL
LIN {X 0,Y 126.366,Z 533.633,A -85,B 0,C 180,E1 -25097.145,E2 -25097.145} C_VEL
LIN {X 0,Y 126.245,Z 532.629,A -85,B 0,C 180,E1 -25100.384,E2 -25100.384} C_VEL
LIN {X 0,Y 126.783,Z 529.779,A -85,B 0,C 180,E1 -25106.194,E2 -25106.194} C_VEL
LIN {X 0,Y 127.697,Z 525.777,A -85,B 0,C 180,E1 -25111.575,E2 -25111.575} C_VEL
LIN {X 0,Y 129.263,Z 521.079,A -85,B 0,C 180,E1 -25116.241,E2 -25116.241} C_VEL
LIN {X 0,Y 131.834,Z 514.031,A -85,B 0,C 180,E1 -25121.53,E2 -25121.53} C_VEL
LIN {X 0,Y 134.82,Z 506.385,A -85,B 0,C 180,E1 -25125.881,E2 -25125.881} C_VEL
LIN {X 0,Y 138.486,Z 496.774,A -85,B 0,C 180,E1 -25130.031,E2 -25130.031} C_VEL
LIN {X 0,Y 142.031,Z 486.857,A -85,B 0,C 180,E1 -25133.317,E2 -25133.317} C_VEL
LIN {X 0,Y 145.666,Z 475.637,A -85,B 0,C 180,E1 -25136.118,E2 -25136.118} C_VEL
LIN {X 0,Y 148.71,Z 464.643,A -85,B 0,C 180,E1 -25138.201,E2 -25138.201} C_VEL
LIN {X 0,Y 151.081,Z 452.587,A -85,B 0,C 180,E1 -25140.002,E2 -25140.002} C_VEL
LIN {X 0,Y 152.929,Z 439.872,A -85,B 0,C 180,E1 -25141.34,E2 -25141.34} C_VEL
LIN {X 0,Y 154.442,Z 426.926,A -85,B 0,C 180,E1 -25142.112,E2 -25142.112} C_VEL
LIN {X 0,Y 157.247,Z 381.755,A -85,B 0,C 180,E1 -25143.938,E2 -25143.938} C_VEL
LIN {X 0,Y 151.768,Z 370.059,A -85,B 0,C 180,E1 -25146.404,E2 -25146.404} C_VEL
LIN {X 0,Y 145.983,Z 359.511,A -85,B 0,C 180,E1 -25149.206,E2 -25149.206} C_VEL
LIN {X 0,Y 140.345,Z 350.984,A -85,B 0,C 180,E1 -25152.182,E2 -25152.182} C_VEL
LIN {X 0,Y 138.279,Z 347.977,A -85,B 0,C 180,E1 -25153.368,E2 -25153.368} C_VEL
LIN {X 0,Y 135.648,Z 344.261,A -85,B 0,C 180,E1 -25154.966,E2 -25154.966} C_VEL
LIN {X 0,Y 133.221,Z 341.184,A -85,B 0,C 180,E1 -25156.515,E2 -25156.515} C_VEL
LIN {X 0,Y 132.423,Z 339.683,A -85,B 0,C 180,E1 -25157.093,E2 -25157.093} C_VEL
LIN {X 0,Y 130.061,Z 337.481,A -85,B 0,C 180,E1 -25158.681,E2 -25158.681} C_VEL
LIN {X 0,Y 129.066,Z 335.187,A -85,B 0,C 180,E1 -25159.518,E2 -25159.518} C_VEL
LIN {X 0,Y 128.933,Z 334.403,A -85,B 0,C 180,E1 -25159.737,E2 -25159.737} C_VEL
LIN {X 0,Y 128.953,Z 334.418,A -85,B 0,C 180,E1 -25164.832,E2 -25164.832} C_VEL
LIN {X 0,Y 129.012,Z 334.384,A -85,B 0,C 180,E1 -25170.641,E2 -25170.641} C_VEL
LIN {X 0,Y 129.022,Z 334.413,A -85,B 0,C 180,E1 -25174.166,E2 -25174.166} C_VEL
LIN {X 0,Y 129.102,Z 334.379,A -85,B 0,C 180,E1 -25177.728,E2 -25177.728} C_VEL
LIN {X 0,Y 129.179,Z 334.393,A -85,B 0,C 180,E1 -25184.215,E2 -25184.215} C_VEL
LIN {X 0,Y 129.384,Z 334.345,A -85,B 0,C 180,E1 -25187.877,E2 -25187.877} C_VEL
LIN {X 0,Y 129.46,Z 334.324,A -85,B 0,C 180,E1 -25190.627,E2 -25190.627} C_VEL
LIN {X 0,Y 130.081,Z 334.247,A -85,B 0,C 180,E1 -25200,E2 -25200} C_VEL
LIN {X 0,Y 129.51,Z 334.325,A -85,B 0,C 180,E1 -25209.37,E2 -25209.37} C_VEL
LIN {X 0,Y 129.388,Z 334.341,A -85,B 0,C 180,E1 -25212.549,E2 -25212.549} C_VEL
LIN {X 0,Y 129.149,Z 334.394,A -85,B 0,C 180,E1 -25219.057,E2 -25219.057} C_VEL
LIN {X 0,Y 129.104,Z 334.398,A -85,B 0,C 180,E1 -25222.4,E2 -25222.4} C_VEL
LIN {X 0,Y 129.032,Z 334.411,A -85,B 0,C 180,E1 -25229.375,E2 -25229.375} C_VEL
LIN {X 0,Y 129.018,Z 334.412,A -85,B 0,C 180,E1 -25229.862,E2 -25229.862} C_VEL
LIN {X 0,Y 129.901,Z 337.068,A -85,B 0,C 180,E1 -25230.68,E2 -25230.68} C_VEL
LIN {X 0,Y 131.792,Z 339.175,A -85,B 0,C 180,E1 -25232.001,E2 -25232.001} C_VEL
LIN {X 0,Y 132.776,Z 339.973,A -85,B 0,C 180,E1 -25232.632,E2 -25232.632} C_VEL
LIN {X 0,Y 134.714,Z 343.199,A -85,B 0,C 180,E1 -25233.963,E2 -25233.963} C_VEL
LIN {X 0,Y 136.507,Z 345.305,A -85,B 0,C 180,E1 -25235.056,E2 -25235.056} C_VEL
LIN {X 0,Y 140.464,Z 351.176,A -85,B 0,C 180,E1 -25237.386,E2 -25237.386} C_VEL
LIN {X 0,Y 143.823,Z 356.359,A -85,B 0,C 180,E1 -25239.204,E2 -25239.204} C_VEL
LIN {X 0,Y 149.218,Z 367.621,A -85,B 0,C 180,E1 -25242.044,E2 -25242.044} C_VEL
LIN {X 0,Y 153.79,Z 379.526,A -85,B 0,C 180,E1 -25244.349,E2 -25244.349} C_VEL
LIN {X 0,Y 155.653,Z 385.064,A -85,B 0,C 180,E1 -25245.269,E2 -25245.269} C_VEL
LIN {X 0,Y 156.433,Z 398.034,A -85,B 0,C 180,E1 -25246.265,E2 -25246.265} C_VEL
LIN {X 0,Y 153.681,Z 440.419,A -85,B 0,C 180,E1 -25248.028,E2 -25248.028} C_VEL
LIN {X 0,Y 151.874,Z 454.064,A -85,B 0,C 180,E1 -25249.053,E2 -25249.053} C_VEL
LIN {X 0,Y 149.52,Z 466.073,A -85,B 0,C 180,E1 -25250.398,E2 -25250.398} C_VEL
LIN {X 0,Y 146.944,Z 476.47,A -85,B 0,C 180,E1 -25251.994,E2 -25251.994} C_VEL
LIN {X 0,Y 143.867,Z 486.985,A -85,B 0,C 180,E1 -25254.114,E2 -25254.114} C_VEL
LIN {X 0,Y 140.655,Z 496.735,A -85,B 0,C 180,E1 -25256.661,E2 -25256.661} C_VEL
LIN {X 0,Y 137.163,Z 506.672,A -85,B 0,C 180,E1 -25260.031,E2 -25260.031} C_VEL
LIN {X 0,Y 133.911,Z 515.307,A -85,B 0,C 180,E1 -25263.792,E2 -25263.792} C_VEL
LIN {X 0,Y 131.169,Z 522.763,A -85,B 0,C 180,E1 -25267.974,E2 -25267.974} C_VEL
LIN {X 0,Y 128.789,Z 529.091,A -85,B 0,C 180,E1 -25272.536,E2 -25272.536} C_VEL
LIN {X 0,Y 127.361,Z 534.129,A -85,B 0,C 180,E1 -25277.25,E2 -25277.25} C_VEL
LIN {X 0,Y 126.646,Z 538.01,A -85,B 0,C 180,E1 -25282.027,E2 -25282.027} C_VEL
LIN {X 0,Y 126.468,Z 540.835,A -85,B 0,C 180,E1 -25286.816,E2 -25286.816} C_VEL
LIN {X 0,Y 126.515,Z 542.402,A -85,B 0,C 180,E1 -25290.717,E2 -25290.717} C_VEL
LIN {X 0,Y 126.47,Z 543.562,A -85,B 0,C 180,E1 -25296.383,E2 -25296.383} C_VEL
LIN {X 0,Y 127.146,Z 543.476,A -85,B 0,C 180,E1 -25301.293,E2 -25301.293} C_VEL
LIN {X 0,Y 128.471,Z 542.645,A -85,B 0,C 180,E1 -25305.876,E2 -25305.876} C_VEL
LIN {X 0,Y 129.786,Z 541.576,A -85,B 0,C 180,E1 -25308.961,E2 -25308.961} C_VEL
LIN {X 0,Y 133.312,Z 538.524,A -85,B 0,C 180,E1 -25314.328,E2 -25314.328} C_VEL
LIN {X 0,Y 134.577,Z 536.861,A -85,B 0,C 180,E1 -25316.695,E2 -25316.695} C_VEL
LIN {X 0,Y 135.362,Z 533.647,A -85,B 0,C 180,E1 -25320.671,E2 -25320.671} C_VEL
LIN {X 0,Y 136.638,Z 529.737,A -85,B 0,C 180,E1 -25324.481,E2 -25324.481} C_VEL
LIN {X 0,Y 138.6,Z 526.986,A -85,B 0,C 180,E1 -25326.503,E2 -25326.503} C_VEL
LIN {X 0,Y 144.476,Z 520.278,A -85,B 0,C 180,E1 -25330.133,E2 -25330.133} C_VEL
LIN {X 0,Y 150.86,Z 512.069,A -85,B 0,C 180,E1 -25333.406,E2 -25333.406} C_VEL
LIN {X 0,Y 156.565,Z 503.689,A -85,B 0,C 180,E1 -25335.909,E2 -25335.909} C_VEL
LIN {X 0,Y 162.538,Z 493.375,A -85,B 0,C 180,E1 -25338.235,E2 -25338.235} C_VEL
LIN {X 0,Y 167.505,Z 483.195,A -85,B 0,C 180,E1 -25339.972,E2 -25339.972} C_VEL
LIN {X 0,Y 172.092,Z 472.069,A -85,B 0,C 180,E1 -25341.357,E2 -25341.357} C_VEL
LIN {X 0,Y 176.053,Z 459.675,A -85,B 0,C 180,E1 -25342.506,E2 -25342.506} C_VEL
LIN {X 0,Y 179.002,Z 446.545,A -85,B 0,C 180,E1 -25343.358,E2 -25343.358} C_VEL
LIN {X 0,Y 180.891,Z 433.051,A -85,B 0,C 180,E1 -25343.905,E2 -25343.905} C_VEL
LIN {X 0,Y 182.167,Z 417.957,A -85,B 0,C 180,E1 -25344.379,E2 -25344.379} C_VEL
LIN {X 0,Y 178.702,Z 408.671,A -85,B 0,C 180,E1 -25347.027,E2 -25347.027} C_VEL
LIN {X 0,Y 175.439,Z 400.987,A -85,B 0,C 180,E1 -25349.755,E2 -25349.755} C_VEL
LIN {X 0,Y 172.12,Z 393.778,A -85,B 0,C 180,E1 -25352.9,E2 -25352.9} C_VEL
LIN {X 0,Y 170.234,Z 390.088,A -85,B 0,C 180,E1 -25354.903,E2 -25354.903} C_VEL
LIN {X 0,Y 168.239,Z 386.154,A -85,B 0,C 180,E1 -25357.308,E2 -25357.308} C_VEL
LIN {X 0,Y 165.894,Z 382.332,A -85,B 0,C 180,E1 -25360.59,E2 -25360.59} C_VEL
LIN {X 0,Y 163.8,Z 379.587,A -85,B 0,C 180,E1 -25364.285,E2 -25364.285} C_VEL
LIN {X 0,Y 163.086,Z 377.758,A -85,B 0,C 180,E1 -25366.13,E2 -25366.13} C_VEL
LIN {X 0,Y 161.273,Z 376.024,A -85,B 0,C 180,E1 -25373.466,E2 -25373.466} C_VEL
LIN {X 0,Y 161.514,Z 375.88,A -85,B 0,C 180,E1 -25378.753,E2 -25378.753} C_VEL
LIN {X 0,Y 163.381,Z 377.96,A -85,B 0,C 180,E1 -25385.09,E2 -25385.09} C_VEL
LIN {X 0,Y 165.027,Z 381.238,A -85,B 0,C 180,E1 -25388.572,E2 -25388.572} C_VEL
LIN {X 0,Y 166.339,Z 382.877,A -85,B 0,C 180,E1 -25390.618,E2 -25390.618} C_VEL
LIN {X 0,Y 169.127,Z 387.295,A -85,B 0,C 180,E1 -25394.284,E2 -25394.284} C_VEL
LIN {X 0,Y 172.011,Z 391.901,A -85,B 0,C 180,E1 -25397.364,E2 -25397.364} C_VEL
LIN {X 0,Y 175.009,Z 396.826,A -85,B 0,C 180,E1 -25400.111,E2 -25400.111} C_VEL
LIN {X 0,Y 179.26,Z 404.434,A -85,B 0,C 180,E1 -25403.503,E2 -25403.503} C_VEL
LIN {X 0,Y 182.615,Z 411.199,A -85,B 0,C 180,E1 -25405.898,E2 -25405.898} C_VEL
LIN {X 0,Y 180.594,Z 432.843,A -85,B 0,C 180,E1 -25406.63,E2 -25406.63} C_VEL
LIN {X 0,Y 178.234,Z 446.294,A -85,B 0,C 180,E1 -25407.397,E2 -25407.397} C_VEL
LIN {X 0,Y 175.004,Z 458.445,A -85,B 0,C 180,E1 -25408.385,E2 -25408.385} C_VEL
LIN {X 0,Y 171.088,Z 470.029,A -85,B 0,C 180,E1 -25409.78,E2 -25409.78} C_VEL
LIN {X 0,Y 166.664,Z 480.322,A -85,B 0,C 180,E1 -25411.359,E2 -25411.359} C_VEL
LIN {X 0,Y 161.254,Z 490.95,A -85,B 0,C 180,E1 -25413.535,E2 -25413.535} C_VEL
LIN {X 0,Y 155.761,Z 499.933,A -85,B 0,C 180,E1 -25415.913,E2 -25415.913} C_VEL
LIN {X 0,Y 149.326,Z 508.859,A -85,B 0,C 180,E1 -25419.051,E2 -25419.051} C_VEL
LIN {X 0,Y 143.22,Z 516.285,A -85,B 0,C 180,E1 -25422.601,E2 -25422.601} C_VEL
LIN {X 0,Y 137.683,Z 522.196,A -85,B 0,C 180,E1 -25426.44,E2 -25426.44} C_VEL
LIN {X 0,Y 132.791,Z 526.809,A -85,B 0,C 180,E1 -25430.571,E2 -25430.571} C_VEL
LIN {X 0,Y 128.561,Z 530.341,A -85,B 0,C 180,E1 -25435.084,E2 -25435.084} C_VEL
LIN {X 0,Y 125.159,Z 532.716,A -85,B 0,C 180,E1 -25439.642,E2 -25439.642} C_VEL
LIN {X 0,Y 123.31,Z 533.783,A -85,B 0,C 180,E1 -25442.872,E2 -25442.872} C_VEL
LIN {X 0,Y 120.698,Z 534.695,A -85,B 0,C 180,E1 -25449.55,E2 -25449.55} C_VEL
LIN {X 0,Y 119.856,Z 534.558,A -85,B 0,C 180,E1 -25452.95,E2 -25452.95} C_VEL
LIN {X 0,Y 119.326,Z 533.98,A -85,B 0,C 180,E1 -25456.372,E2 -25456.372} C_VEL
LIN {X 0,Y 119.144,Z 533.006,A -85,B 0,C 180,E1 -25459.805,E2 -25459.805} C_VEL
LIN {X 0,Y 119.713,Z 529.989,A -85,B 0,C 180,E1 -25466.385,E2 -25466.385} C_VEL
LIN {X 0,Y 120.605,Z 526.314,A -85,B 0,C 180,E1 -25471.668,E2 -25471.668} C_VEL
LIN {X 0,Y 122.189,Z 521.691,A -85,B 0,C 180,E1 -25476.604,E2 -25476.604} C_VEL
LIN {X 0,Y 124.907,Z 514.72,A -85,B 0,C 180,E1 -25482.179,E2 -25482.179} C_VEL
LIN {X 0,Y 128.03,Z 507.182,A -85,B 0,C 180,E1 -25486.748,E2 -25486.748} C_VEL
LIN {X 0,Y 131.18,Z 499.475,A -85,B 0,C 180,E1 -25490.378,E2 -25490.378} C_VEL
LIN {X 0,Y 135.183,Z 489,A -85,B 0,C 180,E1 -25494.166,E2 -25494.166} C_VEL
LIN {X 0,Y 138.859,Z 478.331,A -85,B 0,C 180,E1 -25497.096,E2 -25497.096} C_VEL
LIN {X 0,Y 142.058,Z 467.975,A -85,B 0,C 180,E1 -25499.243,E2 -25499.243} C_VEL
LIN {X 0,Y 144.848,Z 455.667,A -85,B 0,C 180,E1 -25501.233,E2 -25501.233} C_VEL
LIN {X 0,Y 146.929,Z 442.661,A -85,B 0,C 180,E1 -25502.774,E2 -25502.774} C_VEL
LIN {X 0,Y 148.597,Z 430.38,A -85,B 0,C 180,E1 -25503.626,E2 -25503.626} C_VEL
LIN {X 0,Y 151.703,Z 384.943,A -85,B 0,C 180,E1 -25505.497,E2 -25505.497} C_VEL
LIN {X 0,Y 151.518,Z 383.519,A -85,B 0,C 180,E1 -25505.647,E2 -25505.647} C_VEL
LIN {X 0,Y 146.148,Z 372.076,A -85,B 0,C 180,E1 -25508.291,E2 -25508.291} C_VEL
LIN {X 0,Y 140.986,Z 362.898,A -85,B 0,C 180,E1 -25511.018,E2 -25511.018} C_VEL
LIN {X 0,Y 135.317,Z 354.021,A -85,B 0,C 180,E1 -25514.337,E2 -25514.337} C_VEL
LIN {X 0,Y 132.064,Z 349.604,A -85,B 0,C 180,E1 -25516.424,E2 -25516.424} C_VEL
LIN {X 0,Y 129.116,Z 345.452,A -85,B 0,C 180,E1 -25518.515,E2 -25518.515} C_VEL
LIN {X 0,Y 126.802,Z 342.694,A -85,B 0,C 180,E1 -25520.256,E2 -25520.256} C_VEL
LIN {X 0,Y 125.668,Z 340.74,A -85,B 0,C 180,E1 -25521.225,E2 -25521.225} C_VEL
LIN {X 0,Y 123.3,Z 338.746,A -85,B 0,C 180,E1 -25523.164,E2 -25523.164} C_VEL
LIN {X 0,Y 122.119,Z 336.41,A -85,B 0,C 180,E1 -25524.358,E2 -25524.358} C_VEL
LIN {X 0,Y 121.905,Z 335.295,A -85,B 0,C 180,E1 -25524.71,E2 -25524.71} C_VEL
LIN {X 0,Y 121.922,Z 335.264,A -85,B 0,C 180,E1 -25529.838,E2 -25529.838} C_VEL
LIN {X 0,Y 121.977,Z 335.283,A -85,B 0,C 180,E1 -25536.214,E2 -25536.214} C_VEL
LIN {X 0,Y 122.025,Z 335.25,A -85,B 0,C 180,E1 -25539.784,E2 -25539.784} C_VEL
LIN {X 0,Y 122.233,Z 335.248,A -85,B 0,C 180,E1 -25546.704,E2 -25546.704} C_VEL
LIN {X 0,Y 122.398,Z 335.202,A -85,B 0,C 180,E1 -25550.081,E2 -25550.081} C_VEL
LIN {X 0,Y 122.588,Z 335.21,A -85,B 0,C 180,E1 -25556.714,E2 -25556.714} C_VEL
LIN {X 0,Y 123.035,Z 335.124,A -85,B 0,C 180,E1 -25560,E2 -25560} C_VEL
LIN {X 0,Y 122.44,Z 335.232,A -85,B 0,C 180,E1 -25566.592,E2 -25566.592} C_VEL
LIN {X 0,Y 122.44,Z 335.201,A -85,B 0,C 180,E1 -25569.916,E2 -25569.916} C_VEL
LIN {X 0,Y 122.257,Z 335.234,A -85,B 0,C 180,E1 -25573.294,E2 -25573.294} C_VEL
LIN {X 0,Y 122.042,Z 335.284,A -85,B 0,C 180,E1 -25580.214,E2 -25580.214} C_VEL
LIN {X 0,Y 121.988,Z 335.371,A -85,B 0,C 180,E1 -25584.916,E2 -25584.916} C_VEL
LIN {X 0,Y 122.826,Z 337.874,A -85,B 0,C 180,E1 -25585.868,E2 -25585.868} C_VEL
LIN {X 0,Y 124.727,Z 340.079,A -85,B 0,C 180,E1 -25587.534,E2 -25587.534} C_VEL
LIN {X 0,Y 126.1,Z 341.142,A -85,B 0,C 180,E1 -25588.609,E2 -25588.609} C_VEL
LIN {X 0,Y 128.123,Z 344.411,A -85,B 0,C 180,E1 -25590.263,E2 -25590.263} C_VEL
LIN {X 0,Y 129.755,Z 346.026,A -85,B 0,C 180,E1 -25591.422,E2 -25591.422} C_VEL
LIN {X 0,Y 132.3,Z 349.75,A -85,B 0,C 180,E1 -25593.218,E2 -25593.218} C_VEL
LIN {X 0,Y 133.737,Z 351.825,A -85,B 0,C 180,E1 -25594.17,E2 -25594.17} C_VEL
LIN {X 0,Y 136.319,Z 355.65,A -85,B 0,C 180,E1 -25595.792,E2 -25595.792} C_VEL
LIN {X 0,Y 139.869,Z 361.304,A -85,B 0,C 180,E1 -25597.877,E2 -25597.877} C_VEL
LIN {X 0,Y 144.957,Z 372.371,A -85,B 0,C 180,E1 -25600.77,E2 -25600.77} C_VEL
